NETWORK
TITLE = ---- ---- Recoger el Atributo de las UTs - PILA (La Carga es una Pila)
/////////////////////////////////////////////////////////////////////////
/////////////////////////////////////////////////////////////////////////
/////////////////////////////////////////////////////////////////////////
AtributoDeUTs_PILA:NOP   0;
      +AR2  P#5.0;

      OPN   DB [#DBEventosRec];
      L     DBB [AR2, P#0.0];  // Sacar el Valor del Campo
      T     #Leido;
      +AR2  P#1.0;

      L     #Leido;  // Comparar si es cero
      L     '0';  // La Carga No es Pila
      ==I;
      JC    InicioBucleAtributos_EventosDeLasUTs;

      SET;
      S     #AtributosDeUTs.AtributosTipoDeCarga.Pila;


// Continuo con el Evento
      JU    InicioBucleAtributos_EventosDeLasUTs;



NETWORK
TITLE = ---- ---- Recoger el Atributo de las UTs - VACI ( La carga esta vacia de contenido)
/////////////////////////////////////////////////////////////////////////
/////////////////////////////////////////////////////////////////////////
/////////////////////////////////////////////////////////////////////////
AtributoDeUTs_VACI:NOP   0;
      +AR2  P#5.0;

      OPN   DB [#DBEventosRec];
      L     DBB [AR2, P#0.0];  // Sacar el Valor del Campo
      T     #Leido;
      +AR2  P#1.0;

      L     #Leido;  // Comparar si es cero
      L     '0';  // La carga No esta Vacia
      ==I;
      JC    InicioBucleAtributos_EventosDeLasUTs;

      SET;
      S     #AtributosDeUTs.AtributosTipoDeCarga.Vacia;


// Continuo con el Evento
      JU    InicioBucleAtributos_EventosDeLasUTs;



NETWORK
TITLE = ---- ---- Recoger el Atributo de las UTs - COTA ( Cota de Altura)
/////////////////////////////////////////////////////////////////////////
/////////////////////////////////////////////////////////////////////////
/////////////////////////////////////////////////////////////////////////
AtributoDeUTs_COTA:NOP   0;
      +AR2  P#5.0;
      TAR2;
      T     #P_Eventos;
      SRD   3;
      T     #OffsetInicial;

// Obtener el Valor del Atributo
      CALL  "FC892_Obtener_ValorDelAtributo"
      ( DB_String := #DBEventosRec,
        OffsetIni := #OffsetInicial,
        Valor     := #ValorDeAtributo
      );

      L     #ValorDeAtributo;  // Lo guardo
      T     #AtributosDeUTs.CotaAltura;

// Continuo con el Evento
      L     #P_Eventos;
      LAR2;
      JU    InicioBucleAtributos_EventosDeLasUTs;



NETWORK
TITLE = ---- ---- Recoger el Atributo de las UTs - COTW (Cota de Anchura)
/////////////////////////////////////////////////////////////////////////
/////////////////////////////////////////////////////////////////////////
/////////////////////////////////////////////////////////////////////////
AtributoDeUTs_COTW:NOP   0;
      +AR2  P#5.0;
      TAR2;
      T     #P_Eventos;
      SRD   3;
      T     #OffsetInicial;

// Obtener el Valor del Atributo
      CALL  "FC892_Obtener_ValorDelAtributo"
      ( DB_String := #DBEventosRec,
        OffsetIni := #OffsetInicial,
        Valor     := #ValorDeAtributo
      );

      L     #ValorDeAtributo;  // Lo guardo
      T     #AtributosDeUTs.CotaAnchura;

// Continuo con el Evento
      L     #P_Eventos;
      LAR2;
      JU    InicioBucleAtributos_EventosDeLasUTs;



NETWORK
TITLE = ---- ---- Recoger el Atributo de las UTs - COTL (Cota de Profundidad)
/////////////////////////////////////////////////////////////////////////
/////////////////////////////////////////////////////////////////////////
/////////////////////////////////////////////////////////////////////////
AtributoDeUTs_COTL:NOP   0;
      +AR2  P#5.0;
      TAR2;
      T     #P_Eventos;
      SRD   3;
      T     #OffsetInicial;

// Obtener el Valor del Atributo
      CALL  "FC892_Obtener_ValorDelAtributo"
      ( DB_String := #DBEventosRec,
        OffsetIni := #OffsetInicial,
        Valor     := #ValorDeAtributo
      );

      L     #ValorDeAtributo;  // Lo guardo
      T     #AtributosDeUTs.CotaProfundidad;

// Continuo con el Evento
      L     #P_Eventos;
      LAR2;
      JU    InicioBucleAtributos_EventosDeLasUTs;



NETWORK
TITLE = ---- ---- Recoger el Atributo de las UTs - PESO
/////////////////////////////////////////////////////////////////////////
/////////////////////////////////////////////////////////////////////////
/////////////////////////////////////////////////////////////////////////
AtributoDeUTs_PESO:NOP   0;
      +AR2  P#5.0;
      TAR2;
      T     #P_Eventos;
      SRD   3;
      T     #OffsetInicial;

// Obtener el Valor del Atributo
      CALL  "FC892_Obtener_ValorDelAtributo"
      ( DB_String := #DBEventosRec,
        OffsetIni := #OffsetInicial,
        Valor     := #ValorDeAtributo
      );

      L     #ValorDeAtributo;  // Lo guardo
      T     #AtributosDeUTs.Peso;

// Continuo con el Evento
      L     #P_Eventos;
      LAR2;
      JU    InicioBucleAtributos_EventosDeLasUTs;



NETWORK
TITLE = ---- ---- Recoger el Atributo de las UTs - ALTO (Codigo de Altura)
/////////////////////////////////////////////////////////////////////////
/////////////////////////////////////////////////////////////////////////
/////////////////////////////////////////////////////////////////////////
AtributoDeUTs_ALTO:NOP   0;
      +AR2  P#5.0;
      TAR2;
      T     #P_Eventos;
      SRD   3;
      T     #OffsetInicial;

// Obtener el Valor del Atributo
      CALL  "FC892_Obtener_ValorDelAtributo"
      ( DB_String := #DBEventosRec,
        OffsetIni := #OffsetInicial,
        Valor     := #ValorDeAtributo
      );

      L     #ValorDeAtributo;  // Lo guardo
      T     #AtributosDeUTs.GaliboAltura;

// Continuo con el Evento
      L     #P_Eventos;
      LAR2;
      JU    InicioBucleAtributos_EventosDeLasUTs;



NETWORK
TITLE = ---- ---- Recoger el Atributo de las UTs - ANCH (Codigo de Anchura)
/////////////////////////////////////////////////////////////////////////
/////////////////////////////////////////////////////////////////////////
/////////////////////////////////////////////////////////////////////////
AtributoDeUTs_ANCH:NOP   0;
      +AR2  P#5.0;
      TAR2;
      T     #P_Eventos;
      SRD   3;
      T     #OffsetInicial;

// Obtener el Valor del Atributo
      CALL  "FC892_Obtener_ValorDelAtributo"
      ( DB_String := #DBEventosRec,
        OffsetIni := #OffsetInicial,
        Valor     := #ValorDeAtributo
      );

      L     #ValorDeAtributo;  // Lo guardo
      T     #AtributosDeUTs.GaliboAnchura;

// Continuo con el Evento
      L     #P_Eventos;
      LAR2;
      JU    InicioBucleAtributos_EventosDeLasUTs;



NETWORK
TITLE = ---- ---- Recoger el Atributo de las UTs - PROF (Codigo de Profundidad)
/////////////////////////////////////////////////////////////////////////
/////////////////////////////////////////////////////////////////////////
/////////////////////////////////////////////////////////////////////////
AtributoDeUTs_PROF:NOP   0;
      +AR2  P#5.0;
      TAR2;
      T     #P_Eventos;
      SRD   3;
      T     #OffsetInicial;

// Obtener el Valor del Atributo
      CALL  "FC892_Obtener_ValorDelAtributo"
      ( DB_String := #DBEventosRec,
        OffsetIni := #OffsetInicial,
        Valor     := #ValorDeAtributo
      );

      L     #ValorDeAtributo;  // Lo guardo
      T     #AtributosDeUTs.GaliboProfundidad;

// Continuo con el Evento
      L     #P_Eventos;
      LAR2;
      JU    InicioBucleAtributos_EventosDeLasUTs;



NETWORK
TITLE = ---- ---- Recoger el Atributo de las UTs - TACO (Codigo de Taco)
/////////////////////////////////////////////////////////////////////////
/////////////////////////////////////////////////////////////////////////
/////////////////////////////////////////////////////////////////////////
AtributoDeUTs_TACO:NOP   0;
      +AR2  P#5.0;
      TAR2;
      T     #P_Eventos;
      SRD   3;
      T     #OffsetInicial;

// Obtener el Valor del Atributo
      CALL  "FC892_Obtener_ValorDelAtributo"
      ( DB_String := #DBEventosRec,
        OffsetIni := #OffsetInicial,
        Valor     := #ValorDeAtributo
      );

      L     #ValorDeAtributo;  // Lo guardo
      T     #AtributosDeUTs.GaliboTaco;

// Continuo con el Evento
      L     #P_Eventos;
      LAR2;
      JU    InicioBucleAtributos_EventosDeLasUTs;



NETWORK
TITLE = ---- ---- Recoger el Atributo de las UTs - HUEC (Codigo de Hueco)
/////////////////////////////////////////////////////////////////////////
/////////////////////////////////////////////////////////////////////////
/////////////////////////////////////////////////////////////////////////
AtributoDeUTs_HUEC:NOP   0;
      +AR2  P#5.0;
      TAR2;
      T     #P_Eventos;
      SRD   3;
      T     #OffsetInicial;

// Obtener el Valor del Atributo
      CALL  "FC892_Obtener_ValorDelAtributo"
      ( DB_String := #DBEventosRec,
        OffsetIni := #OffsetInicial,
        Valor     := #ValorDeAtributo
      );

      L     #ValorDeAtributo;  // Lo guardo
      T     #AtributosDeUTs.GaliboHueco;

// Continuo con el Evento
      L     #P_Eventos;
      LAR2;
      JU    InicioBucleAtributos_EventosDeLasUTs;



NETWORK
TITLE = ---- ---- Recoger el Atributo de las UTs - HUER (Codigo de Hueco de Remontada)
/////////////////////////////////////////////////////////////////////////
/////////////////////////////////////////////////////////////////////////
/////////////////////////////////////////////////////////////////////////
AtributoDeUTs_HUER:NOP   0;
      +AR2  P#5.0;
      TAR2;
      T     #P_Eventos;
      SRD   3;
      T     #OffsetInicial;

// Obtener el Valor del Atributo
      CALL  "FC892_Obtener_ValorDelAtributo"
      ( DB_String := #DBEventosRec,
        OffsetIni := #OffsetInicial,
        Valor     := #ValorDeAtributo
      );

      L     #ValorDeAtributo;  // Lo guardo
      T     #AtributosDeUTs.GaliboHuecoRemontada;

// Continuo con el Evento
      L     #P_Eventos;
      LAR2;
      JU    InicioBucleAtributos_EventosDeLasUTs;



NETWORK
TITLE = ---- ---- Recoger el Atributo de las UTs - COLO (Codigo de Color)
/////////////////////////////////////////////////////////////////////////
/////////////////////////////////////////////////////////////////////////
/////////////////////////////////////////////////////////////////////////
AtributoDeUTs_COLO:NOP   0;
      +AR2  P#5.0;

      OPN   DB [#DBEventosRec];
      L     DBD [AR2, P#0.0];
      T     #EtiquetaAtributo;

// Obtener el Valor del Atributo
      CALL  "FC894_Obtener_ValorDeEtiqueta"
      ( EtiquetaEvento := #EtiquetaAtributo,
        ValorEvento    := #ValorDeEtiqueta
      );

      L     #ValorDeEtiqueta;  // Lo guardo
      T     #AtributosDeUTs.GaliboColor;

// Continuo con el Evento
      +AR2  P#4.0;
      JU    InicioBucleAtributos_EventosDeLasUTs;



NETWORK
TITLE = ---- ---- Recoger el Atributo de las UTs - PATI (Codigo de Patin)
/////////////////////////////////////////////////////////////////////////
/////////////////////////////////////////////////////////////////////////
/////////////////////////////////////////////////////////////////////////
AtributoDeUTs_PATI:NOP   0;
      +AR2  P#5.0;
      TAR2;
      T     #P_Eventos;
      SRD   3;
      T     #OffsetInicial;

// Obtener el Valor del Atributo
      CALL  "FC892_Obtener_ValorDelAtributo"
      ( DB_String := #DBEventosRec,
        OffsetIni := #OffsetInicial,
        Valor     := #ValorDeAtributo
      );

      L     #ValorDeAtributo;  // Lo guardo
      T     #AtributosDeUTs.GaliboPatin;

// Continuo con el Evento
      L     #P_Eventos;
      LAR2;
      JU    InicioBucleAtributos_EventosDeLasUTs;



NETWORK
TITLE = ---- ---- Recoger el Atributo de las UTs - LETI (Lado de la Etiqueta)
/////////////////////////////////////////////////////////////////////////
/////////////////////////////////////////////////////////////////////////
/////////////////////////////////////////////////////////////////////////
AtributoDeUTs_LETI:NOP   0;
      +AR2  P#5.0;
      TAR2;
      T     #P_Eventos;
      SRD   3;
      T     #OffsetInicial;

// Obtener el Valor del Atributo
      CALL  "FC892_Obtener_ValorDelAtributo"
      ( DB_String := #DBEventosRec,
        OffsetIni := #OffsetInicial,
        Valor     := #ValorDeAtributo
      );

      L     #ValorDeAtributo;  // Lo guardo
      L     1;
      +I;
      T     #AtributosDeUTs.PosicionDeLaEtiqueta;

// Continuo con el Evento
      L     #P_Eventos;
      LAR2;
      JU    InicioBucleAtributos_EventosDeLasUTs;



NETWORK
TITLE = ---- ---- Recoger el Atributo de las UTs - SGAP ( SGA - Error de Peso)
/////////////////////////////////////////////////////////////////////////
/////////////////////////////////////////////////////////////////////////
/////////////////////////////////////////////////////////////////////////
AtributoDeUTs_SGAP:NOP   0;
      +AR2  P#5.0;

      OPN   DB [#DBEventosRec];
      L     DBW [AR2, P#0.0];
      T     #Leido;

      L     0;  // Por defecto No Error
      T     #ValorDeAtributo;

      L     'NO';  // Tiene Error ?
      L     #Leido;
      ==I;
      JC    AtributoDeUTs_SGAP_NoError;

      L     W#16#08;
      T     #ValorDeAtributo;

AtributoDeUTs_SGAP_NoError:NOP   0;
      L     #ValorDeAtributo;
      L     #AtributosDeUTs.GaliboSGA;
      +I;
      T     #AtributosDeUTs.GaliboSGA;

// Continuo con el Evento
      +AR2  P#2.0;
      JU    InicioBucleAtributos_EventosDeLasUTs;



NETWORK
TITLE = ---- ---- Recoger el Atributo de las UTs - SGAE ( SGA - Error de Etiqueta)
/////////////////////////////////////////////////////////////////////////
/////////////////////////////////////////////////////////////////////////
/////////////////////////////////////////////////////////////////////////
AtributoDeUTs_SGAE:NOP   0;
      +AR2  P#5.0;

      OPN   DB [#DBEventosRec];
      L     DBW [AR2, P#0.0];
      T     #Leido;

      L     0;  // Por defecto No Error
      T     #ValorDeAtributo;

      L     'NO';  // Tiene Error ?
      L     #Leido;
      ==I;
      JC    AtributoDeUTs_SGAE_NoError;

      L     W#16#04;
      T     #ValorDeAtributo;

AtributoDeUTs_SGAE_NoError:NOP   0;
      L     #ValorDeAtributo;
      L     #AtributosDeUTs.GaliboSGA;
      +I;
      T     #AtributosDeUTs.GaliboSGA;

// Continuo con el Evento
      +AR2  P#2.0;
      JU    InicioBucleAtributos_EventosDeLasUTs;



NETWORK
TITLE = ---- ---- Recoger el Atributo de las UTs - SGAD ( SGA - Error de Dimensiones)
/////////////////////////////////////////////////////////////////////////
/////////////////////////////////////////////////////////////////////////
/////////////////////////////////////////////////////////////////////////
AtributoDeUTs_SGAD:NOP   0;
      +AR2  P#5.0;

      OPN   DB [#DBEventosRec];
      L     DBW [AR2, P#0.0];
      T     #Leido;

      L     0;  // Por defecto No Error
      T     #ValorDeAtributo;

      L     'NO';  // Tiene Error ?
      L     #Leido;
      ==I;
      JC    AtributoDeUTs_SGAD_NoError;

      L     W#16#02;
      T     #ValorDeAtributo;

AtributoDeUTs_SGAD_NoError:NOP   0;
      L     #ValorDeAtributo;
      L     #AtributosDeUTs.GaliboSGA;
      +I;
      T     #AtributosDeUTs.GaliboSGA;

// Continuo con el Evento
      +AR2  P#2.0;
      JU    InicioBucleAtributos_EventosDeLasUTs;



NETWORK
TITLE = ---- ---- Recoger el Atributo de las UTs - SGA_ ( SGA - Error General)
/////////////////////////////////////////////////////////////////////////
/////////////////////////////////////////////////////////////////////////
/////////////////////////////////////////////////////////////////////////
AtributoDeUTs_SGA_Error:NOP   0;
      +AR2  P#5.0;

      OPN   DB [#DBEventosRec];
      L     DBW [AR2, P#0.0];
      T     #Leido;

      L     0;  // Por defecto No Error
      T     #ValorDeAtributo;

      L     'NO';  // Tiene Error ?
      L     #Leido;
      ==I;
      JC    AtributoDeUTs_SGA_Error_NoError;

      L     W#16#01;
      T     #ValorDeAtributo;

AtributoDeUTs_SGA_Error_NoError:NOP   0;
      L     #ValorDeAtributo;
      L     #AtributosDeUTs.GaliboSGA;
      +I;
      T     #AtributosDeUTs.GaliboSGA;

// Continuo con el Evento
      +AR2  P#2.0;
      JU    InicioBucleAtributos_EventosDeLasUTs;



NETWORK
TITLE = ---- ---- Recoger el Atributo de las UTs - RSLT (Mover UT - Resultado)
/////////////////////////////////////////////////////////////////////////
/////////////////////////////////////////////////////////////////////////
/////////////////////////////////////////////////////////////////////////
AtributoDeUTs_RSLT:NOP   0;
      +AR2  P#5.0;

      OPN   DB [#DBEventosRec];
      L     DBW [AR2, P#0.0];  // Sacar el Valor del Campo
      T     #Leido;

      SET;  // Inicializar a NOK
      S     #AtributosDeUTs.CambiarUTDeMesa.NOK;
      R     #AtributosDeUTs.CambiarUTDeMesa.OK;

      L     #Leido;  // Comparar si es NO ?
      L     'SI';
      <>I;
      JC    InicioBucleAtributos_EventosDeLasUTs;

      SET;  // Inicializar a OK
      R     #AtributosDeUTs.CambiarUTDeMesa.NOK;
      S     #AtributosDeUTs.CambiarUTDeMesa.OK;

// Continuo con el Evento
      +AR2  P#2.0;
      JU    InicioBucleAtributos_EventosDeLasUTs;



NETWORK
TITLE = ---- ---- Recoger el Atributo de las UTs - PDST (Mover UT - Posicion en la Cola de Mesa)
/////////////////////////////////////////////////////////////////////////
/////////////////////////////////////////////////////////////////////////
/////////////////////////////////////////////////////////////////////////
AtributoDeUTs_PDST:NOP   0;
      +AR2  P#5.0;

      OPN   DB [#DBEventosRec];
      L     DBD [AR2, P#0.0];  // Sacar el Valor del Campo
      T     #EtiquetaAtributo;

      SET;  // Inicializar a Final
      S     #AtributosDeUTs.CambiarUTDeMesa.Final;
      R     #AtributosDeUTs.CambiarUTDeMesa.Inicio;

      L     #EtiquetaAtributo;  // Comparar si es _FIN ?
      L     '_INI';
      <>D;
      JC    InicioBucleAtributos_EventosDeLasUTs;

      SET;  // Inicializar a Inicio
      R     #AtributosDeUTs.CambiarUTDeMesa.Final;
      S     #AtributosDeUTs.CambiarUTDeMesa.Inicio;

// Continuo con el Evento
      +AR2  P#4.0;
      JU    InicioBucleAtributos_EventosDeLasUTs;



NETWORK
TITLE = ---- ---- Recoger el Atributo de las UTs - DEST (Mover UT - Destino)
/////////////////////////////////////////////////////////////////////////
/////////////////////////////////////////////////////////////////////////
/////////////////////////////////////////////////////////////////////////
AtributoDeUTs_DEST:NOP   0;
      +AR2  P#5.0;
      TAR2;
      T     #P_Eventos;
      SRD   3;
      T     #OffsetInicial;

// Obtener el Valor del Atributo
      CALL  "FC892_Obtener_ValorDelAtributo"
      ( DB_String := #DBEventosRec,
        OffsetIni := #OffsetInicial,
        Valor     := #ValorDeAtributo
      );

      L     #ValorDeAtributo;  // Lo guardo
      L     #AtributosDeUTs.CambiarUTDeMesa.Destino;

// Continuo con el Evento
      L     #P_Eventos;
      LAR2;
      JU    InicioBucleAtributos_EventosDeLasUTs;



NETWORK
TITLE = ////////////////////////////////////////////////////////////////////////////////////////////////////////////

NETWORK
TITLE = Analizar la lista de los Atributos de los Dispositivos
Atributos_EventosDeLosDispositivos:NOP   0;

/////////////////////////////////////////////////////////////////////////
/////////////////////////////////////////////////////////////////////////
/////////////////////////////////////////////////////////////////////////
// Inicializa variables de los Atributos de las UTs
      L     0;
      T     #Cero;

      CALL  FILL
      ( BVAL    := #Cero,
        RET_VAL := #ReturnValor,
        BLK     := #AtributosDeDispositivos
      );  // Inicializa Atributos de las UTS



NETWORK
TITLE = ----
/////////////////////////////////////////////////////////////////////////
/////////////////////////////////////////////////////////////////////////
// Buscando Atributos o Final del Evento
      +AR2  P#4.0;  // Prepara Puntero para ver los atributos

InicioBucleAtributos_EventosDeLosDispositivos:NOP   0;
      OPN   DB [#DBEventosRec];
      L     DBB [AR2, P#0.0];
      T     #Leido;

// Inicio de atributo - Ir a tratar los atributos
      L     #Leido;
      L     '[';  // '[' - Inicio de Atributo
      ==I;  // Atributo del Evento
      JC    EncontradoAtributos_EventosDeLosDispositivos;

// Fin del Evento
      L     #Leido;
      L     '}';  // '}' - Fin del Evento
      ==I;  // Se acabo el evento
      JC    FinalAtributos_EventosDeLosDispositivos;

      +AR2  P#1.0;  // Seguir buscado atributo
      JU    InicioBucleAtributos_EventosDeLosDispositivos;


/////////////////////////////////////////////////////////////////////////
/////////////////////////////////////////////////////////////////////////
// Se acaba el Evento - Ir a guardar datos del Evento
FinalAtributos_EventosDeLosDispositivos:NOP   0;
      TAR2;
      T     #P_Eventos;  // Guardo Por donde voy en la lista de eventos
      JU    GuardarDatos_EventosRecibidos;



NETWORK
TITLE = Distribucion de los Atributos de los DIspositivos (LIsta del DB de Conversion)
EncontradoAtributos_EventosDeLosDispositivos:NOP   0;

/////////////////////////////////////////////////////////////////////////
/////////////////////////////////////////////////////////////////////////
/////////////////////////////////////////////////////////////////////////
/////////////////////////////////////////////////////////////////////////
// Mirar que Atributo del Evento  es ?
      +AR2  P#1.0;
      OPN   DB [#DBEventosRec];
      L     DBD [AR2, P#0.0];  // Atributo - 4 Caracteres
      T     #Atributo;

/////////////////////////////////////////////////////////////////////////
/////////////////////////////////////////////////////////////////////////
/////////////////////////////////////////////////////////////////////////
// Buscar numero de Atributo
      L     1;
      T     #NumeroAtributo;
BucleDeBusqueda_NumeroDeAtributoDeDispositivos:NOP   0;

// -- Se ha encontrado el Atributo Recibido
      L     "DB870_ConversorEventos".AtributosRecibidosDeDispositivos[#NumeroAtributo];
      L     #Atributo;
      ==D;
      JC    Encontrado_NumeroDeAtributoDeDispositivos;

// -- Final de la lista de Atributo Recibidos - No Encontrado
      L     "DB870_ConversorEventos".AtributosRecibidosDeDispositivos[#NumeroAtributo];
      L     0;
      ==D;
      JC    InicioBucleAtributos_EventosDeLosDispositivos;

// --- Maximo del Array de la Lista de Atributo Recibidos - No Encontrado
      L     #NumeroAtributo;
      L     "CTE_MaxArrayConversion";
      >=I;
      JC    InicioBucleAtributos_EventosDeLosDispositivos;


// --- Continuar la Busqueda
      L     #NumeroAtributo;
      L     1;
      +I;
      T     #NumeroAtributo;
      JU    BucleDeBusqueda_NumeroDeAtributoDeDispositivos;



NETWORK
TITLE = ----
/////////////////////////////////////////////////////////////////////////
/////////////////////////////////////////////////////////////////////////
/////////////////////////////////////////////////////////////////////////
// Distribuir dependiendo del Resultado de la Busqueda de Atributo Recibido
Encontrado_NumeroDeAtributoDeDispositivos:NOP   0;
      L     #NumeroAtributo;
      JL    NoExiste_NumeroDeAtibutoDeDispositivos;

      JU    NoExiste_NumeroDeAtibutoDeDispositivos;
      JU    AtributoDeDispositivos_TIPO;  // Atributo (01) - TIPO
      JU    AtributoDeDispositivos_NUME;  // Atributo (02) - NUME
      JU    AtributoDeDispositivos_NUES;  // Atributo (03) - NUES
      JU    AtributoDeDispositivos_HABI;  // Atributo (04) - HABI
      JU    AtributoDeDispositivos_PRIO;  // Atributo (05) - PRIO

      JU    AtributoDeDispositivos_SONO;  // Atributo (06) - SONO
      JU    AtributoDeDispositivos_VERD;  // Atributo (07) - VERD
      JU    AtributoDeDispositivos_ROJO;  // Atributo (08) - ROJO
      JU    AtributoDeDispositivos_AMAR;  // Atributo (09) - AMAR
      JU    AtributoDeDispositivos_AZUL;  // Atributo (10) - AZUL

      JU    AtributoDeDispositivos_MOTI;  // Atributo (11) - MOTI
      JU    AtributoDeDispositivos_OPER;  // Atributo (12) - OPER
      JU    AtributoDeDispositivos_TEXT;  // Atributo (13) - TEXT

      JU    AtributoDeDispositivos_HORQ;  // Atributo (14) - HORQ
      JU    AtributoDeDispositivos_POSI;  // Atributo (15) - POSI

/////////////////////////////////////////////////////////////////////////
NoExiste_NumeroDeAtibutoDeDispositivos:NOP   0;
      JU    InicioBucleAtributos_EventosDeLosDispositivos;



NETWORK
TITLE = ---- ---- Recoger el Atributo de los Dispositivos - TIPO
/////////////////////////////////////////////////////////////////////////
/////////////////////////////////////////////////////////////////////////
/////////////////////////////////////////////////////////////////////////
AtributoDeDispositivos_TIPO:NOP   0;
      +AR2  P#5.0;

      OPN   DB [#DBEventosRec];
      L     DBD [AR2, P#0.0];
      T     #EtiquetaAtributo;

// Obtener el Valor del Tipo de Dispositivo

      CALL  "FC894_Obtener_ValorDeEtiqueta"
      ( EtiquetaEvento := #EtiquetaAtributo,
        ValorEvento    := #ValorDeEtiqueta
      );

      L     #ValorDeEtiqueta;  // Lo guardo
      T     #AtributosDeDispositivos.Tipo;

// Continuo con el Evento
      +AR2  P#4.0;
      JU    InicioBucleAtributos_EventosDeLosDispositivos;



NETWORK
TITLE = ---- ---- Recoger el Atributo de los Dispositivos - NUME
/////////////////////////////////////////////////////////////////////////
/////////////////////////////////////////////////////////////////////////
/////////////////////////////////////////////////////////////////////////
AtributoDeDispositivos_NUME:NOP   0;
      +AR2  P#5.0;
      TAR2;
      T     #P_Eventos;
      SRD   3;
      T     #OffsetInicial;

// Obtener el Valor del Numero del Dispositivo

      CALL  "FC892_Obtener_ValorDelAtributo"
      ( DB_String := #DBEventosRec,
        OffsetIni := #OffsetInicial,
        Valor     := #ValorDeAtributo
      );
      L     #ValorDeAtributo;  // Lo guardo
      T     #AtributosDeDispositivos.Numero;

// Continuo con el Evento
      L     #P_Eventos;
      LAR2;
      JU    InicioBucleAtributos_EventosDeLosDispositivos;



NETWORK
TITLE = ---- ---- Recoger el Atributo de los Dispositivos - NUES (Nuevo Estado)
/////////////////////////////////////////////////////////////////////////
/////////////////////////////////////////////////////////////////////////
/////////////////////////////////////////////////////////////////////////
AtributoDeDispositivos_NUES:NOP   0;
      +AR2  P#5.0;

      OPN   DB [#DBEventosRec];
      L     DBD [AR2, P#0.0];
      T     #EtiquetaAtributo;

// Obtener el Valor del Tipo de Dispositivo
      CALL  "FC894_Obtener_ValorDeEtiqueta"
      ( EtiquetaEvento := #EtiquetaAtributo,
        ValorEvento    := #ValorDeEtiqueta
      );

      L     #ValorDeEtiqueta;  // Lo guardo
      T     #AtributosDeDispositivos.NuevoEstado;

// Continuo con el Evento
      +AR2  P#4.0;
      JU    InicioBucleAtributos_EventosDeLosDispositivos;



NETWORK
TITLE = ---- ---- Recoger el Atributo de los Dispositivos - HABI
/////////////////////////////////////////////////////////////////////////
/////////////////////////////////////////////////////////////////////////
/////////////////////////////////////////////////////////////////////////
AtributoDeDispositivos_HABI:NOP   0;
      +AR2  P#5.0;

      OPN   DB [#DBEventosRec];
      L     DBW [AR2, P#0.0];
      T     #Leido;

      L     2001;
      T     #ValorDeAtributo;

      L     #Leido;
      L     'NO';
      ==I;
      JCN   AtributoDeDispositivos_HABI_NoHabilitar;

      L     2002;
      T     #ValorDeAtributo;

AtributoDeDispositivos_HABI_NoHabilitar:NOP   0;
      L     #ValorDeAtributo;  // Lo guardo
      T     #AtributosDeDispositivos.Habilitado;

// Continuo con el Evento
      +AR2  P#2.0;
      JU    InicioBucleAtributos_EventosDeLosDispositivos;



NETWORK
TITLE = ---- ---- Recoger el Atributo de los Dispositivos - PRIO
/////////////////////////////////////////////////////////////////////////
/////////////////////////////////////////////////////////////////////////
/////////////////////////////////////////////////////////////////////////
AtributoDeDispositivos_PRIO:NOP   0;
      +AR2  P#5.0;
      TAR2;
      T     #P_Eventos;
      SRD   3;
      T     #OffsetInicial;

// Obtener el Valor del Numero del Dispositivo
      CALL  "FC892_Obtener_ValorDelAtributo"
      ( DB_String := #DBEventosRec,
        OffsetIni := #OffsetInicial,
        Valor     := #ValorDeAtributo
      );

      L     #ValorDeAtributo;  // Lo guardo
      L     1;
      +I;
      T     #AtributosDeDispositivos.Prioridad;

// Continuo con el Evento
      L     #P_Eventos;
      LAR2;
      JU    InicioBucleAtributos_EventosDeLosDispositivos;



NETWORK
TITLE = ---- ---- Recoger el Atributo de los Dispositivos - SONO (Baliza - Sirena)
/////////////////////////////////////////////////////////////////////////
/////////////////////////////////////////////////////////////////////////
/////////////////////////////////////////////////////////////////////////
AtributoDeDispositivos_SONO:NOP   0;
      +AR2  P#5.0;

      SET;
      S     #AtributosDeDispositivos.BalizaColor.Sonoro;


// Continuo con el Evento
      JU    InicioBucleAtributos_EventosDeLosDispositivos;



NETWORK
TITLE = ---- ---- Recoger el Atributo de los Dispositivos - VERD (Baliza - Verde)
/////////////////////////////////////////////////////////////////////////
/////////////////////////////////////////////////////////////////////////
/////////////////////////////////////////////////////////////////////////
AtributoDeDispositivos_VERD:NOP   0;
      +AR2  P#5.0;

      SET;
      S     #AtributosDeDispositivos.BalizaColor.Verde;


// Continuo con el Evento
      JU    InicioBucleAtributos_EventosDeLosDispositivos;



NETWORK
TITLE = ---- ---- Recoger el Atributo de los Dispositivos - ROJO (Baliza - Roja)
/////////////////////////////////////////////////////////////////////////
/////////////////////////////////////////////////////////////////////////
/////////////////////////////////////////////////////////////////////////
AtributoDeDispositivos_ROJO:NOP   0;
      +AR2  P#5.0;

      SET;
      S     #AtributosDeDispositivos.BalizaColor.Rojo;


// Continuo con el Evento
      JU    InicioBucleAtributos_EventosDeLosDispositivos;



NETWORK
TITLE = ---- ---- Recoger el Atributo de los Dispositivos - AMAR (Baliza - Amarilla)
/////////////////////////////////////////////////////////////////////////
/////////////////////////////////////////////////////////////////////////
/////////////////////////////////////////////////////////////////////////
AtributoDeDispositivos_AMAR:NOP   0;
      +AR2  P#5.0;

      SET;
      S     #AtributosDeDispositivos.BalizaColor.Amarillo;


// Continuo con el Evento
      JU    InicioBucleAtributos_EventosDeLosDispositivos;



NETWORK
TITLE = ---- ---- Recoger el Atributo de los Dispositivos - AZUL (Baliza - Azul)
/////////////////////////////////////////////////////////////////////////
/////////////////////////////////////////////////////////////////////////
/////////////////////////////////////////////////////////////////////////
AtributoDeDispositivos_AZUL:NOP   0;
      +AR2  P#5.0;

      SET;
      S     #AtributosDeDispositivos.BalizaColor.Azul;


// Continuo con el Evento
      JU    InicioBucleAtributos_EventosDeLosDispositivos;



NETWORK
TITLE = ---- ---- Recoger el Atributo de los Dispositivos - MOTI (Moitvo del Envio a Error del JdT )
/////////////////////////////////////////////////////////////////////////
/////////////////////////////////////////////////////////////////////////
/////////////////////////////////////////////////////////////////////////
AtributoDeDispositivos_MOTI:NOP   0;
      +AR2  P#5.0;

// - Recorrer el Motivo del Error es una STRING
      L     2;  // Inicializaciones
      T     #LonguitudTextoRecibido;

// Inicio a Recoger el Motivo del Error
AtributoDeDispositivos_MOTI_InicioBucle:NOP   0;
      OPN   DB [#DBEventosRec];
      L     DBB [AR2, P#0.0];  // Leer ek texto
      T     #Leido;

      L     #Leido;  // Es final del Texto
      L     '[';
      ==I;
      JC    AtributoDeDispositivos_MOTI_FinalBucle;

      L     #Leido;  // Es final del Texto
      L     '}';
      ==I;
      JC    AtributoDeDispositivos_MOTI_FinalBucle;

      L     #Leido;  // Guardo el texto
      T     #AtributosDeDispositivos.MotivoDelError[#LonguitudTextoRecibido];

// Incremetar punteros
      +AR2  P#1.0;
      L     #LonguitudTextoRecibido;
      L     1;
      +I;
      T     #LonguitudTextoRecibido;

      L     0;  // Pongo el siguiente a cero
      T     #AtributosDeDispositivos.MotivoDelError[#LonguitudTextoRecibido];

      JU    AtributoDeDispositivos_MOTI_InicioBucle;


// - Continuo con el Evento
AtributoDeDispositivos_MOTI_FinalBucle:NOP   0;
      L     48;  // Inicio la carcacteristica de la STRING
      T     #AtributosDeDispositivos.MotivoDelError[0];
      L     #LonguitudTextoRecibido;
      L     2;
      -I;
      T     #AtributosDeDispositivos.MotivoDelError[1];

      JU    InicioBucleAtributos_EventosDeLosDispositivos;



NETWORK
TITLE = ---- ---- Recoger el Atributo de los Dispositivos - OPER (Operacion a realizar de las Maquinas)
/////////////////////////////////////////////////////////////////////////
/////////////////////////////////////////////////////////////////////////
/////////////////////////////////////////////////////////////////////////
AtributoDeDispositivos_OPER:NOP   0;
      +AR2  P#5.0;

      OPN   DB [#DBEventosRec];
      L     DBD [AR2, P#0.0];
      T     #EtiquetaAtributo;

// Obtener el Valor del Tipo de Dispositivo
      CALL  "FC894_Obtener_ValorDeEtiqueta"
      ( EtiquetaEvento := #EtiquetaAtributo,
        ValorEvento    := #ValorDeEtiqueta
      );

      L     #ValorDeEtiqueta;  // Lo guardo
      T     #AtributosDeDispositivos.Operacion;

// Continuo con el Evento
      +AR2  P#4.0;
      JU    InicioBucleAtributos_EventosDeLosDispositivos;



NETWORK
TITLE = ---- ---- Recoger el Atributo de los Dispositivos - TEXT
/////////////////////////////////////////////////////////////////////////
/////////////////////////////////////////////////////////////////////////
/////////////////////////////////////////////////////////////////////////
AtributoDeDispositivos_TEXT:NOP   0;
      +AR2  P#5.0;

// - Recorrer el Motivo del Error es una STRING
      L     2;  // Inicializaciones
      T     #LonguitudTextoRecibido;

// Inicio a Recoger el Texto
AtributoDeDispositivos_TEXT_InicioBucle:NOP   0;
      OPN   DB [#DBEventosRec];
      L     DBB [AR2, P#0.0];  // Leer ek texto
      T     #Leido;

      L     #Leido;  // Es final del Texto
      L     '[';
      ==I;
      JC    AtributoDeDispositivos_TEXT_FinalBucle;

      L     #Leido;  // Es final del Texto
      L     '}';
      ==I;
      JC    AtributoDeDispositivos_TEXT_FinalBucle;

      L     #Leido;  // Guardo el texto
      T     #AtributosDeDispositivos.TextoRecibido[#LonguitudTextoRecibido];

// Incremetar punteros
      +AR2  P#1.0;
      L     #LonguitudTextoRecibido;
      L     1;
      +I;
      T     #LonguitudTextoRecibido;

      L     0;  // Pongo el siguiente a cero
      T     #AtributosDeDispositivos.TextoRecibido[#LonguitudTextoRecibido];

      JU    AtributoDeDispositivos_TEXT_InicioBucle;


// - Continuo con el Evento
AtributoDeDispositivos_TEXT_FinalBucle:NOP   0;
      L     48;  // Inicio la carcacteristica de la STRING
      T     #AtributosDeDispositivos.TextoRecibido[0];
      L     #LonguitudTextoRecibido;
      L     2;
      -I;
      T     #AtributosDeDispositivos.TextoRecibido[1];

      JU    InicioBucleAtributos_EventosDeLosDispositivos;



NETWORK
TITLE = ---- ---- Recoger el Atributo de los Dispositivos - HORQ
/////////////////////////////////////////////////////////////////////////
/////////////////////////////////////////////////////////////////////////
/////////////////////////////////////////////////////////////////////////
AtributoDeDispositivos_HORQ:NOP   0;
      +AR2  P#5.0;
      TAR2;
      T     #P_Eventos;
      SRD   3;
      T     #OffsetInicial;

// Obtener el Valor del Numero del Dispositivo
      CALL  "FC892_Obtener_ValorDelAtributo"
      ( DB_String := #DBEventosRec,
        OffsetIni := #OffsetInicial,
        Valor     := #ValorDeAtributo
      );
      L     #ValorDeAtributo;  // Lo guardo
      T     #AtributosDeDispositivos.MesaHorquilla;

// Continuo con el Evento
      L     #P_Eventos;
      LAR2;
      JU    InicioBucleAtributos_EventosDeLosDispositivos;



NETWORK
TITLE = ---- ---- Recoger el Atributo de los Dispositivos - POSI
/////////////////////////////////////////////////////////////////////////
/////////////////////////////////////////////////////////////////////////
/////////////////////////////////////////////////////////////////////////
AtributoDeDispositivos_POSI:NOP   0;
      +AR2  P#5.0;
      TAR2;
      T     #P_Eventos;
      SRD   3;
      T     #OffsetInicial;

// Obtener el Valor del Numero del Dispositivo
      CALL  "FC892_Obtener_ValorDelAtributo"
      ( DB_String := #DBEventosRec,
        OffsetIni := #OffsetInicial,
        Valor     := #ValorDeAtributo
      );
      L     #ValorDeAtributo;  // Lo guardo
      T     #AtributosDeDispositivos.MesaCargaDesCarga;

// Continuo con el Evento
      L     #P_Eventos;
      LAR2;
      JU    InicioBucleAtributos_EventosDeLosDispositivos;



NETWORK
TITLE = Distribucion para Guardar Datos del Evento Recibido (LIsta del DB de Conversion) ///////
/////////////////////////////////////////////////////////////////////////
/////////////////////////////////////////////////////////////////////////
/////////////////////////////////////////////////////////////////////////
GuardarDatos_EventosRecibidos:NOP   0;
      TAR2;
      T     #P_Eventos;  // Guardo Por donde voy en la lista de eventos

      L     #NumeroEvento;
      JL    NoExiste_GuardarDatos_Eventos;

      JU    NoExiste_GuardarDatos_Eventos;
      JU    GuardarDatos_EventoRecibido_CREA;  // Evento (01) - CREA
      JU    GuardarDatos_EventoRecibido_RUTA;  // Evento (02) - RUTA
      JU    GuardarDatos_EventoRecibido_DRUT;  // Evento (03) - DRUT
      JU    GuardarDatos_EventoRecibido_RETI;  // Evento (04) - RETI
      JU    GuardarDatos_EventoRecibido_BORR;  // Evento (05) - BORR
      JU    GuardarDatos_EventoRecibido_DATA;  // Evento (06) - DATA
      JU    GuardarDatos_EventoRecibido_Refresco_UT;  // Evento (07) - ?UT?
      JU    GuardarDatos_EventoRecibido_MOVE;  // Evento (08) - MOVE
      JU    GuardarDatos_EventoRecibido_DEMB;  // Evento (09) - DEMB

      JU    GuardarDatos_EventoRecibido_CSTA;  // Evento (10) - CSTA
      JU    GuardarDatos_EventoRecibido_DIDO;  // Evento (11) - DIDO

      JU    NoExiste_GuardarDatos_Eventos;  // Evento (12) - ORDE
      JU    NoExiste_GuardarDatos_Eventos;  // Evento (13) - BOET
      JU    NoExiste_GuardarDatos_Eventos;  // Evento (14) - BOBD
      JU    NoExiste_GuardarDatos_Eventos;  // Evento (15) - RUET
      JU    NoExiste_GuardarDatos_Eventos;  // Evento (16) - RUES
      JU    NoExiste_GuardarDatos_Eventos;  // Evento (17) - INIR

      JU    GuardarDatos_EventoRecibido_Refresco_ST;  // Evento (18) - ?ST?

      JU    NoExiste_GuardarDatos_Eventos;  // Evento (19) - QCRE
      JU    NoExiste_GuardarDatos_Eventos;  // Evento (20) - QPR?

      JU    NoExiste_GuardarDatos_Eventos;  // Evento (21) - CHEQ

/////////////////////////////////////////////////////////////////////////
NoExiste_GuardarDatos_Eventos:NOP   0;
      L     #P_Eventos;  // Recupero por donde voy en la lista de eventos
      LAR2;  // Regreso a buscar el siguiente evento
      JU    FinBucle_EventosRecibidos;



NETWORK
TITLE = ////////////////////////////////////////////////////////////////////////////////////////////////////////////

NETWORK
TITLE = Guardar Datos - Evento CREA - Crear una Nueva UT
// Analisis del evento
//   - Inicializa variables de los atributos del Evento
//   - Buscar Atributos o Final del Evento
//   - Guardar datos del Evento
// Analisis de los atributos del Evento
//   - Mirar que atributo del Evento es
//   - Distribuir a recoger los datos del Evento
//   - Recoger el Atributo McKey
//   - Recoger el Atributo MesaActual
//   - Recoger el Atributo Tipo
//   - Recoger el Atributo Codigo de Barras
//   - Recoger el Atributo Grupo de UT
//   - Recoger el Atributo Cantidad de UT en el Grupo
//   - Recoger el Atributo Orden dentro del grupo
//   - Recoger el Atributo Altura
GuardarDatos_EventoRecibido_CREA:NOP   0;

/////////////////////////////////////////////////////////////////////////
/////////////////////////////////////////////////////////////////////////
/////////////////////////////////////////////////////////////////////////
// --- Guardar Datos del Evento Recibido


/////////////////////////////////////////////////////////////////////////
/////////////////////////////////////////////////////////////////////////
/////////////////////////////////////////////////////////////////////////
// --- Control de la Mesa Actual es correcta
      L     #AtributosDeUTs.MesaActual;  // Ver que mesa es
      L     "CTE_OffsetMesa";
      -I;
      T     #VarTempUTs.MesaActual;

      L     #VarTempUTs.MesaActual;  // Comprobar el numero de mesa
      L     1;  // No menor de 1
      <I;  // No es correcto
      JC    Final_EventoRecibido_CREA;
      L     #VarTempUTs.MesaActual;
      L     "CTE_MaxMesas";  // No mayor que el parametro
      >I;  // No es correcto
      JC    Final_EventoRecibido_CREA;


/////////////////////////////////////////////////////////////////////////
/////////////////////////////////////////////////////////////////////////
/////////////////////////////////////////////////////////////////////////
// --- Control del Mckey es correcto
      L     #AtributosDeUTs.Mckey;  // Se ha recibido Mckey = 0
      L     0;  // No se puede Crear
      ==D;
      JC    Final_EventoRecibido_CREA;


/////////////////////////////////////////////////////////////////////////
/////////////////////////////////////////////////////////////////////////
/////////////////////////////////////////////////////////////////////////
// --- Control del Nuevo Mckey no este en el sistema
// --- Comprobación de DUPLICIDAD
      CALL  "FC720_BuscarUT_EnMesa"
      ( Mckey      := #AtributosDeUTs.Mckey,
        MesaActual := #VarTempUTs.MesaActual,
        NumeroUT   := #VarTempUTs.NumeroUT
      );

      L     #VarTempUTs.NumeroUT;  // Existe UT, Hay DUPLICIDAD de Mckey
      L     0;
      ==I;
      JC    MckeyCorrecto_EventoRecibido_CREA;

// --- Informe de Duplicadad del Mckey
      SET;
      S     "DB812_UTs_Control".UT[#VarTempUTs.NumeroUT].EventosInformarJdT.DuplicidadMckey;

      JU    Final_EventoRecibido_CREA;

MckeyCorrecto_EventoRecibido_CREA:NOP   0;


/////////////////////////////////////////////////////////////////////////
/////////////////////////////////////////////////////////////////////////
/////////////////////////////////////////////////////////////////////////
// --- Control de la Mesa este Definida
      SET;
      AN    "DB850_DefinicionMesas".Mesa[#VarTempUTs.MesaActual].ConfigMesa.MesaPaso;
      AN    "DB850_DefinicionMesas".Mesa[#VarTempUTs.MesaActual].ConfigMesa.MesaCruce;
      AN    "DB850_DefinicionMesas".Mesa[#VarTempUTs.MesaActual].ConfigMesa.MesaMultiplesDestinos;
      JC    Final_EventoRecibido_CREA;


/////////////////////////////////////////////////////////////////////////
/////////////////////////////////////////////////////////////////////////
/////////////////////////////////////////////////////////////////////////
// --- Crear UT en la Mesa Actual
// --- Nota: Rellena ya en UT el Mckey y la Mesa Actual
      CALL  "FC721_CrearUT_EnMesa"
      ( McKey      := #AtributosDeUTs.Mckey,
        MesaActual := #VarTempUTs.MesaActual,
        NumeroUT   := #VarTempUTs.NumeroUT
      );

      L     #VarTempUTs.NumeroUT;
      L     0;  // No se ha podido crear
      ==I;
      JC    Final_EventoRecibido_CREA;



NETWORK
TITLE = ---- Accion del Evento
/////////////////////////////////////////////////////////////////////////
/////////////////////////////////////////////////////////////////////////
/////////////////////////////////////////////////////////////////////////
// --- Guardar datos en la UT, Mckey y Mesa ya estan
      L     202;  // 202 - Recibido Evento de Creada una Nueva UT en la Mesa
      T     "DB812_UTs_Control".UT[#VarTempUTs.NumeroUT].EstadoEventoRecibido;

      L     #AtributosDeUTs.TipoCarga;
      T     "DB812_UTs_Control".UT[#VarTempUTs.NumeroUT].TipoCarga;

      SET;
      A     #AtributosDeUTs.AtributosTipoDeCarga.Pila;
      S     "DB812_UTs_Control".UT[#VarTempUTs.NumeroUT].AtributosDelaCarga.Pila;
      SET;
      A     #AtributosDeUTs.AtributosTipoDeCarga.Remontada;
      S     "DB812_UTs_Control".UT[#VarTempUTs.NumeroUT].AtributosDelaCarga.Remontada;
      SET;
      A     #AtributosDeUTs.AtributosTipoDeCarga.Vacia;
      S     "DB812_UTs_Control".UT[#VarTempUTs.NumeroUT].AtributosDelaCarga.Vacia;


      L     #AtributosDeUTs.GaliboAltura;
      T     "DB815_UTs_Datos".UT[#VarTempUTs.NumeroUT].GaliboAltura;
      L     #AtributosDeUTs.GaliboAnchura;
      T     "DB815_UTs_Datos".UT[#VarTempUTs.NumeroUT].GaliboAnchura;
      L     #AtributosDeUTs.GaliboProfundidad;
      T     "DB815_UTs_Datos".UT[#VarTempUTs.NumeroUT].GaliboProfundidad;

      L     #AtributosDeUTs.GaliboTaco;
      T     "DB815_UTs_Datos".UT[#VarTempUTs.NumeroUT].GaliboTaco;
      L     #AtributosDeUTs.GaliboHueco;
      T     "DB815_UTs_Datos".UT[#VarTempUTs.NumeroUT].GaliboHueco;
      L     #AtributosDeUTs.GaliboHuecoRemontada;
      T     "DB815_UTs_Datos".UT[#VarTempUTs.NumeroUT].GaliboHuecoRemontado;

      L     #AtributosDeUTs.GaliboColor;
      T     "DB815_UTs_Datos".UT[#VarTempUTs.NumeroUT].GaliboColor;
      L     #AtributosDeUTs.GaliboPatin;
      T     "DB815_UTs_Datos".UT[#VarTempUTs.NumeroUT].GaliboPatin;


      L     #AtributosDeUTs.CodigoFlejado;
      T     "DB815_UTs_Datos".UT[#VarTempUTs.NumeroUT].CodigoFlejado;
      L     #AtributosDeUTs.CodigoEnfardado;
      T     "DB815_UTs_Datos".UT[#VarTempUTs.NumeroUT].CodigoEnfardado;
      L     #AtributosDeUTs.CodigoEtiquetado;
      T     "DB815_UTs_Datos".UT[#VarTempUTs.NumeroUT].CodigoEtiquetado;

      L     #AtributosDeUTs.Peso;
      T     "DB815_UTs_Datos".UT[#VarTempUTs.NumeroUT].Peso;

      L     #AtributosDeUTs.CotaAltura;
      T     "DB815_UTs_Datos".UT[#VarTempUTs.NumeroUT].CotaAltura;
      L     #AtributosDeUTs.CotaAnchura;
      T     "DB815_UTs_Datos".UT[#VarTempUTs.NumeroUT].CotaAnchura;
      L     #AtributosDeUTs.CotaProfundidad;
      T     "DB815_UTs_Datos".UT[#VarTempUTs.NumeroUT].CotaProfundidad;

      L     #AtributosDeUTs.CotaAmarre;
      T     "DB815_UTs_Datos".UT[#VarTempUTs.NumeroUT].Amarre;
      L     #AtributosDeUTs.Presion;
      T     "DB815_UTs_Datos".UT[#VarTempUTs.NumeroUT].Presion;

      L     #AtributosDeUTs.Grupo;
      T     "DB812_UTs_Control".UT[#VarTempUTs.NumeroUT].Grupo;
      L     #AtributosDeUTs.CantidadGrupo;
      T     "DB812_UTs_Control".UT[#VarTempUTs.NumeroUT].CantidadGrupo;
      L     #AtributosDeUTs.PosicionGrupo;
      T     "DB812_UTs_Control".UT[#VarTempUTs.NumeroUT].PosicionGrupo;


/////////////////////////////////////////////////////////////////////////
// --- Posicion de la Etiqueta (0) Derecha (1) Izquierdo
      SET;  // Posicion de la Etiqueta
      L     #AtributosDeUTs.PosicionDeLaEtiqueta;
      L     1;  // Lado Derecho = 0
      ==I;
      R     "DB812_UTs_Control".UT[#VarTempUTs.NumeroUT].AtributosDeLaUT.LadoDeLaEtiqueta;

      SET;  // Posicion de la Etiqueta
      L     #AtributosDeUTs.PosicionDeLaEtiqueta;
      L     2;  // Lado Izquierdo = 1
      ==I;
      S     "DB812_UTs_Control".UT[#VarTempUTs.NumeroUT].AtributosDeLaUT.LadoDeLaEtiqueta;


/////////////////////////////////////////////////////////////////////////
// --- Guardar la etiqueta
      CALL  BLKMOV
      ( SRCBLK  := #AtributosDeUTs.Etiqueta,
        RET_VAL := #ReturnValor,
        DSTBLK  := "DB814_UTs_Etiqueta".UT[#VarTempUTs.NumeroUT].Etiqueta
      );

/////////////////////////////////////////////////////////////////////////
// --- Guardar Datos de QUBIQA
      L     #AtributosDeUTs.QUBIQA_NumeroBulto;  // Numero de Bulto
      T     "DB820_UTs_DatosQUBIQA".UT[#VarTempUTs.NumeroUT].NumeroDeBulto;
      L     #AtributosDeUTs.QUBIQA_TotalBultos;  // Numero de Bultos
      T     "DB820_UTs_DatosQUBIQA".UT[#VarTempUTs.NumeroUT].TotalBultos;

      CALL  BLKMOV
      ( SRCBLK  := #AtributosDeUTs.QUBIQA_PID,
        RET_VAL := #ReturnValor,
        DSTBLK  := "DB820_UTs_DatosQUBIQA".UT[#VarTempUTs.NumeroUT].PID
      );  // Guardar el PID


/////////////////////////////////////////////////////////////////////////
// Guardar Ruta si es necesario
// Si hay ruta Nueva - Guardar MesaDestino, Mesa Intermedia y la nueva ruta
      L     0;  // Si existe Nueva Ruta - MesaDestino <> 0
      L     #AtributosDeUTs.MesaDestino;
      ==I;
      JC    FinalGuardarRuta_EventoRecibido_CREA;


/////////////////////////////////////////////////////////////////////////
// Puntero a la UT, Marcar si es necesario -->
//           Actual = Destino = InterMedia --> Marcar la UT
// MODIFICACION --> 06/05/2013 (Alonso)

      SET;  // Reset - Recircular la Carga - Memoria del Retirar
      R     "DB812_UTs_Control".UT[#VarTempUTs.NumeroUT].AtributosDeLaUT.RecircularCarga;
      R     "DB812_UTs_Control".UT[#VarTempUTs.NumeroUT].AtributosDeLaUT.MemorizarRETI;

      L     "DB812_UTs_Control".UT[#VarTempUTs.NumeroUT].MesaActual;
      L     #AtributosDeUTs.MesaDestino;
      <>I;  // MesaActual <> MesaDestino ?
      JC    NoRecirculaLaCarga_EventoRecibido_CREA;

      L     #AtributosDeUTs.MesaDestino;
      L     #AtributosDeUTs.Ruta[0];
      ==I;
      JC    NoRecirculaLaCarga_EventoRecibido_CREA;

      SET;  // Set - Recircular la Carga
      S     "DB812_UTs_Control".UT[#VarTempUTs.NumeroUT].AtributosDeLaUT.RecircularCarga;

NoRecirculaLaCarga_EventoRecibido_CREA:NOP   0;

      L     #AtributosDeUTs.MesaDestino;
      T     "DB812_UTs_Control".UT[#VarTempUTs.NumeroUT].MesaDestino;
      L     #AtributosDeUTs.MesaIntermedia;
      T     "DB812_UTs_Control".UT[#VarTempUTs.NumeroUT].MesaIntermedia;

      CALL  BLKMOV
      ( SRCBLK  := #AtributosDeUTs.Ruta,
        RET_VAL := #ReturnValor,
        DSTBLK  := "DB813_UTs_Ruta".UT[#VarTempUTs.NumeroUT].Ruta
      );

      L     201;  // 201 - Recibido Evento de nueva ruta para la UT
      T     "DB812_UTs_Control".UT[#VarTempUTs.NumeroUT].EstadoEventoRecibido;

//////////////////////////////////////////////////////////////////////
/// Inicio - Realizado 2017 07 06 // Control para Peticion de Ruta
      L     "DB812_UTs_Control".UT[#VarTempUTs.NumeroUT].MesaActual;
      L     #AtributosDeUTs.MesaDestino;
      <>I;
      JC    FinalGuardarRuta_EventoRecibido_CREA;

// Activar la Peticion de RUTA por llegada a su destino
      L     21;  // 21 - Generar Evento Pedir Ruta
      T     "DB812_UTs_Control".UT[#VarTempUTs.NumeroUT].EstadoGeneralUT;
      L     0;  // 0 - No Vale el Evento Recibido
      T     "DB812_UTs_Control".UT[#VarTempUTs.NumeroUT].EstadoEventoRecibido;

//////////////////////////////////////////////////////////////////////
// Final de Guardar Ruta
FinalGuardarRuta_EventoRecibido_CREA:NOP   0;



NETWORK
TITLE = ---- Final
/////////////////////////////////////////////////////////////////////////
/////////////////////////////////////////////////////////////////////////
/////////////////////////////////////////////////////////////////////////
// Se acabo el evento
Final_EventoRecibido_CREA:NOP   0;
      L     #P_Eventos;  // Recupero por donde voy en la lista de eventos
      LAR2;  // Regreso a buscar el siguiente evento
      JU    FinBucle_EventosRecibidos;



NETWORK
TITLE = Guardar Datos - Evento RUTA - Asignar ruta nueva a la UT
// Analisis del evento
//   - Inicializa variables de los atributos del Evento
//   - Buscar Atributos o Final del Evento
//   - Guardar datos del Evento
// Analisis de los atributos del Evento
//   - Mirar que atributo del Evento es
//   - Distribuir a recoger los datos del Evento
//   - Recoger el Atributo McKey
//   - Recoger el Atributo MesaActual
//   - Recoger el Atributo Nueva Ruta
GuardarDatos_EventoRecibido_RUTA:NOP   0;

/////////////////////////////////////////////////////////////////////////
/////////////////////////////////////////////////////////////////////////
/////////////////////////////////////////////////////////////////////////
// --- Guardar Datos del Evento Recibido


/////////////////////////////////////////////////////////////////////////
/////////////////////////////////////////////////////////////////////////
/////////////////////////////////////////////////////////////////////////
// --- Control de la Mesa Actual es Correcta
      L     #AtributosDeUTs.MesaActual;
      L     0;
      ==I;
      JC    FinControlMesa_EventoRecibido_RUTA;

      L     #AtributosDeUTs.MesaActual;  // Ver que mesa es
      L     "CTE_OffsetMesa";
      -I;
      T     #VarTempUTs.MesaActual;

      L     #VarTempUTs.MesaActual;  // Comprobar el numero de mesa
      L     1;  // No menor de 1
      <I;  // No es correcto
      JC    Final_EventoRecibido_RUTA;
      L     #VarTempUTs.MesaActual;
      L     "CTE_MaxMesas";  // No mayor que el parametro
      >I;  // No es correcto
      JC    Final_EventoRecibido_RUTA;

/////////////////////////////////////////////////////////////////////////
FinControlMesa_EventoRecibido_RUTA:NOP   0;


/////////////////////////////////////////////////////////////////////////
/////////////////////////////////////////////////////////////////////////
/////////////////////////////////////////////////////////////////////////
// --- Buscar UT en la Mesa Actual o por Mckey

      CALL  "FC720_BuscarUT_EnMesa"
      ( Mckey      := #AtributosDeUTs.Mckey,
        MesaActual := #VarTempUTs.MesaActual,
        NumeroUT   := #VarTempUTs.NumeroUT
      );

      L     #VarTempUTs.NumeroUT;
      L     0;
      ==I;  // No existe UT
      JC    Final_EventoRecibido_RUTA;



NETWORK
TITLE = ---- Accion del Evento
/////////////////////////////////////////////////////////////////////////
/////////////////////////////////////////////////////////////////////////
/////////////////////////////////////////////////////////////////////////
// Puntero a la UT, Marcar si es necesario -->
//           Actual = Destino = InterMedia --> Marcar la UT
// MODIFICACION --> 06/05/2013 (Alonso)

      SET;  // Reset - Recircular la Carga - Memoria del Retirar
      R     "DB812_UTs_Control".UT[#VarTempUTs.NumeroUT].AtributosDeLaUT.RecircularCarga;
      R     "DB812_UTs_Control".UT[#VarTempUTs.NumeroUT].AtributosDeLaUT.MemorizarRETI;

      L     "DB812_UTs_Control".UT[#VarTempUTs.NumeroUT].MesaActual;
      L     #AtributosDeUTs.MesaDestino;
      <>I;  // MesaActual <> MesaDestino ?
      JC    GuardarRutaRecibida_EventoRecibido_RUTA;

      L     #AtributosDeUTs.MesaDestino;
      L     #AtributosDeUTs.Ruta[0];
      ==I;
      JC    GuardarRutaRecibida_EventoRecibido_RUTA;

      SET;  // Set - Recircular la Carga
      S     "DB812_UTs_Control".UT[#VarTempUTs.NumeroUT].AtributosDeLaUT.RecircularCarga;


/////////////////////////////////////////////////////////////////////////
/////////////////////////////////////////////////////////////////////////
/////////////////////////////////////////////////////////////////////////
// --- Guardar ruta
GuardarRutaRecibida_EventoRecibido_RUTA:NOP   0;

      L     #AtributosDeUTs.MesaDestino;
      T     "DB812_UTs_Control".UT[#VarTempUTs.NumeroUT].MesaDestino;
      L     #AtributosDeUTs.MesaIntermedia;
      T     "DB812_UTs_Control".UT[#VarTempUTs.NumeroUT].MesaIntermedia;

      CALL  BLKMOV
      ( SRCBLK  := #AtributosDeUTs.Ruta,
        RET_VAL := #ReturnValor,
        DSTBLK  := "DB813_UTs_Ruta".UT[#VarTempUTs.NumeroUT].Ruta
      );

      L     201;  // 201 - Recibido Evento de Nueva Ruta para la UT
      T     "DB812_UTs_Control".UT[#VarTempUTs.NumeroUT].EstadoEventoRecibido;


/////////////////////////////////////////////////////////////////////////
/////////////////////////////////////////////////////////////////////////
//////////////////////////////////////////////////////////////////////
/// Inicio - Realizado 2017 07 06 // Control para Peticion de Ruta
      L     "DB812_UTs_Control".UT[#VarTempUTs.NumeroUT].MesaActual;
      L     #AtributosDeUTs.MesaDestino;
      <>I;
      JC    NoPedirRuta_EventoRecibido_RUTA;

      SET;  // Recircular la Carga ?
      A     "DB812_UTs_Control".UT[#VarTempUTs.NumeroUT].AtributosDeLaUT.RecircularCarga;
      JC    NoPedirRuta_EventoRecibido_RUTA;

// Activar la Peticion de RUTA por llegada a su destino
      L     21;  // 21 - Generar Evento Pedir Ruta
      T     "DB812_UTs_Control".UT[#VarTempUTs.NumeroUT].EstadoGeneralUT;
      L     0;  // 0 - No Vale el Evento Recibido
      T     "DB812_UTs_Control".UT[#VarTempUTs.NumeroUT].EstadoEventoRecibido;

//////////////////////////////////////////////////////////////////////
NoPedirRuta_EventoRecibido_RUTA:NOP   0;



NETWORK
TITLE = ---- Final
//////////////////////////////////////////////////////////////////////
//////////////////////////////////////////////////////////////////////
//////////////////////////////////////////////////////////////////////
// --- Se acabo el evento
Final_EventoRecibido_RUTA:NOP   0;
      L     #P_Eventos;  // Recupero por donde voy en la lista de eventos
      LAR2;  // Regreso a buscar el siguiente evento
      JU    FinBucle_EventosRecibidos;



NETWORK
TITLE = Guardar Datos - Evento DRUT - Asignar ruta nueva a la UT (Dinamica)
// Analisis del evento
//   - Inicializa variables de los atributos del Evento
//   - Buscar Atributos o Final del Evento
//   - Guardar datos del Evento
// Analisis de los atributos del Evento
//   - Mirar que atributo del Evento es
//   - Distribuir a recoger los datos del Evento
//   - Recoger el Atributo McKey
//   - Recoger el Atributo MesaActual
//   - Recoger el Atributo Nueva Ruta
GuardarDatos_EventoRecibido_DRUT:NOP   0;

/////////////////////////////////////////////////////////////////////////
/////////////////////////////////////////////////////////////////////////
/////////////////////////////////////////////////////////////////////////
// --- Guardar Datos del Evento Recibido


/////////////////////////////////////////////////////////////////////////
/////////////////////////////////////////////////////////////////////////
/////////////////////////////////////////////////////////////////////////
// --- Control de la Mesa Actual Recibida
      L     #AtributosDeUTs.MesaActual;
      L     0;
      ==I;
      JC    FinControlMesa_EventoRecibido_DRUT;

      L     #AtributosDeUTs.MesaActual;  // Ver que mesa es
      L     "CTE_OffsetMesa";
      -I;
      T     #VarTempUTs.MesaActual;

      L     #VarTempUTs.MesaActual;  // Comprobar el numero de mesa
      L     1;  // No menor de 1
      <I;  // No es correcto
      JC    Final_EventoRecibido_DRUT;
      L     #VarTempUTs.MesaActual;
      L     "CTE_MaxMesas";  // No mayor que el parametro
      >I;  // No es correcto
      JC    Final_EventoRecibido_DRUT;

/////////////////////////////////////////////////////////////////////////
FinControlMesa_EventoRecibido_DRUT:NOP   0;


/////////////////////////////////////////////////////////////////////////
/////////////////////////////////////////////////////////////////////////
/////////////////////////////////////////////////////////////////////////
// --- Buscar UT en la Mesa Actual o por Mckey

      CALL  "FC720_BuscarUT_EnMesa"
      ( Mckey      := #AtributosDeUTs.Mckey,
        MesaActual := #VarTempUTs.MesaActual,
        NumeroUT   := #VarTempUTs.NumeroUT
      );

      L     #VarTempUTs.NumeroUT;
      L     0;  // No existe UT
      ==I;
      JC    Final_EventoRecibido_DRUT;



NETWORK
TITLE = ---- Accion del Evento
/////////////////////////////////////////////////////////////////////////
/////////////////////////////////////////////////////////////////////////
/////////////////////////////////////////////////////////////////////////
// --- Guardar ruta

      L     #AtributosDeUTs.MesaDestino;
      T     "DB812_UTs_Control".UT[#VarTempUTs.NumeroUT].MesaDestino;
      L     #AtributosDeUTs.MesaIntermedia;
      T     "DB812_UTs_Control".UT[#VarTempUTs.NumeroUT].MesaIntermedia;

      CALL  BLKMOV
      ( SRCBLK  := #AtributosDeUTs.Ruta,
        RET_VAL := #ReturnValor,
        DSTBLK  := "DB813_UTs_Ruta".UT[#VarTempUTs.NumeroUT].Ruta
      );



NETWORK
TITLE = ---- Final
//////////////////////////////////////////////////////////////////////
//////////////////////////////////////////////////////////////////////
//////////////////////////////////////////////////////////////////////
// --- Se acabo el evento
Final_EventoRecibido_DRUT:NOP   0;
      L     #P_Eventos;  // Recupero por donde voy en la lista de eventos
      LAR2;  // Regreso a buscar el siguiente evento
      JU    FinBucle_EventosRecibidos;



NETWORK
TITLE = Guardar Datos - Evento RETI - Retirar la UT
// Analisis del evento
//   - Inicializa variables de los atributos del Evento
//   - Buscar Atributos o Final del Evento
//   - Guardar datos del Evento
// Analisis de los atributos del Evento
//   - Mirar que atributo del Evento es
//   - Distribuir a recoger los datos del Evento
//   - Recoger el Atributo McKey
//   - Recoger el Atributo MesaActual
GuardarDatos_EventoRecibido_RETI:NOP   0;

/////////////////////////////////////////////////////////////////////////
/////////////////////////////////////////////////////////////////////////
/////////////////////////////////////////////////////////////////////////
// --- Guardar Datos del Evento Recibido


/////////////////////////////////////////////////////////////////////////
/////////////////////////////////////////////////////////////////////////
/////////////////////////////////////////////////////////////////////////
// --- Control de Mesa Recibida
      L     #AtributosDeUTs.MesaActual;
      L     0;
      ==I;
      JC    FinControlMesa_EventoRecibido_RETI;

      L     #AtributosDeUTs.MesaActual;  // Ver que mesa es
      L     "CTE_OffsetMesa";
      -I;
      T     #VarTempUTs.MesaActual;

      L     #VarTempUTs.MesaActual;  // Comprobar el numero de mesa
      L     1;  // No menor de 1
      <I;  // No es correcto
      JC    Final_EventoRecibido_RETI;
      L     #VarTempUTs.MesaActual;
      L     "CTE_MaxMesas";  // No mayor que el parametro
      >I;  // No es correcto
      JC    Final_EventoRecibido_RETI;

/////////////////////////////////////////////////////////////////////////
FinControlMesa_EventoRecibido_RETI:NOP   0;


/////////////////////////////////////////////////////////////////////////
/////////////////////////////////////////////////////////////////////////
/////////////////////////////////////////////////////////////////////////
// --- Buscar UT en la Mesa Actual o Mckey
      CALL  "FC720_BuscarUT_EnMesa"
      ( Mckey      := #AtributosDeUTs.Mckey,
        MesaActual := #VarTempUTs.MesaActual,
        NumeroUT   := #VarTempUTs.NumeroUT
      );

      L     #VarTempUTs.NumeroUT;
      L     0;  // No existe UT
      ==I;
      JC    Final_EventoRecibido_RETI;



NETWORK
TITLE = ---- Accion del Evento
/////////////////////////////////////////////////////////////////////////
/////////////////////////////////////////////////////////////////////////
/////////////////////////////////////////////////////////////////////////
// --- Guardar datos
      L     #AtributosDeUTs.OrdenSalida;  // Sumar el numero de salida del Atributo
      L     210;  // 210 - Evento de Retirar la UT por S0
      +I;
      T     #VarTempUTs.SalidaEventoRETI;

      SET;  // Memorizar RETI - Ya memorizado
      A     "DB812_UTs_Control".UT[#VarTempUTs.NumeroUT].AtributosDeLaUT.MemorizarRETI;
      JC    ActivadaMemoria_EventoRecibido_RETI;

      L     #VarTempUTs.SalidaEventoRETI;  // EstadoEventoRecibido
      T     "DB812_UTs_Control".UT[#VarTempUTs.NumeroUT].EstadoEventoRecibido;

/////////////////////////////////////////////////////////////////////////
ActivadaMemoria_EventoRecibido_RETI:NOP   0;

      L     #VarTempUTs.SalidaEventoRETI;  // Mesa Intermeria --> Salida RETI
      T     "DB812_UTs_Control".UT[#VarTempUTs.NumeroUT].MesaIntermedia;

      SET;  // Set - Memorizar RETI
      S     "DB812_UTs_Control".UT[#VarTempUTs.NumeroUT].AtributosDeLaUT.MemorizarRETI;



NETWORK
TITLE = ---- Final
/////////////////////////////////////////////////////////////////////////
/////////////////////////////////////////////////////////////////////////
/////////////////////////////////////////////////////////////////////////
// Se acabo el evento
Final_EventoRecibido_RETI:NOP   0;
      L     #P_Eventos;  // Recupero por donde voy en la lista de eventos
      LAR2;  // Regreso a buscar el siguiente evento
      JU    FinBucle_EventosRecibidos;



NETWORK
TITLE = Guardar Datos - Evento BORR - Borrar la UT
// Analisis del evento
//   - Inicializa variables de los atributos del Evento
//   - Buscar Atributos o Final del Evento
//   - Guardar datos del Evento
// Analisis de los atributos del Evento
//   - Mirar que atributo del Evento es
//   - Distribuir a recoger los datos del Evento
//   - Recoger el Atributo McKey
//   - Recoger el Atributo MesaActual
GuardarDatos_EventoRecibido_BORR:NOP   0;

/////////////////////////////////////////////////////////////////////////
/////////////////////////////////////////////////////////////////////////
/////////////////////////////////////////////////////////////////////////
// --- Guardar Datos del Evento Recibido


/////////////////////////////////////////////////////////////////////////
/////////////////////////////////////////////////////////////////////////
/////////////////////////////////////////////////////////////////////////
// --- Control de Mesa Recibida
      L     #AtributosDeUTs.MesaActual;
      L     0;
      ==I;
      JC    FinControlMesa_EventoRecibido_BORR;

      L     #AtributosDeUTs.MesaActual;  // Ver que mesa es
      L     "CTE_OffsetMesa";
      -I;
      T     #VarTempUTs.MesaActual;

      L     #VarTempUTs.MesaActual;  // Comprobar el numero de mesa
      L     1;  // No menor de 1
      <I;  // No es correcto
      JC    Final_EventoRecibido_BORR;
      L     #VarTempUTs.MesaActual;
      L     "CTE_MaxMesas";  // No mayor que el parametro
      >I;  // No es correcto
      JC    Final_EventoRecibido_BORR;

/////////////////////////////////////////////////////////////////////////
FinControlMesa_EventoRecibido_BORR:NOP   0;



NETWORK
TITLE = ---- Accion del Evento --> Distribucion
/////////////////////////////////////////////////////////////////////////
/////////////////////////////////////////////////////////////////////////
/////////////////////////////////////////////////////////////////////////
// --- Distribucion

      L     0;  // Borrar UT en Particular
      L     #AtributosDeUTs.Mckey;
      <>D;
      JC    BorrarUT_EventoRecibido_BORR;

      L     0;  // Borrar UTs de la Mesa
      L     #AtributosDeUTs.MesaActual;
      <>I;
      JC    BorrarUTsDeMesa_EventoRecibido_BORR;

/////////////////////////////////////////////////////////////////////////
// --- Defecto --> Borrar todas las UTs
      JU    BorrarTodasLasUTs_EventoRecibido_BORR;



NETWORK
TITLE = ---- Accion del Evento --> Borrar UT
/////////////////////////////////////////////////////////////////////////
/////////////////////////////////////////////////////////////////////////
/////////////////////////////////////////////////////////////////////////
// --- Borrar una UT en particular
BorrarUT_EventoRecibido_BORR:NOP   0;
      L     #AtributosDeUTs.MesaActual;
      T     #VarTempUTs.MesaActual;
      L     0;  // Comprobar si hay mesa
      ==I;
      JC    BuscarUT_BorrarUT_EventoRecibido_BORR;

      L     #AtributosDeUTs.MesaActual;  // Ver que mesa es
      L     "CTE_OffsetMesa";
      -I;
      T     #VarTempUTs.MesaActual;

      L     #VarTempUTs.MesaActual;  // Comprobar el numero de mesa
      L     1;  // No menor de 1
      <I;  // No es correcto
      JC    Final_EventoRecibido_BORR;
      L     #VarTempUTs.MesaActual;
      L     "CTE_MaxMesas";  // No mayor que el parametro
      >I;  // No es correcto
      JC    Final_EventoRecibido_BORR;

BuscarUT_BorrarUT_EventoRecibido_BORR:NOP   0;

/////////////////////////////////////////////////////////////////////////
// --- Buscar UT en la Mesa Actual o por Mckey

      CALL  "FC720_BuscarUT_EnMesa"
      ( Mckey      := #AtributosDeUTs.Mckey,
        MesaActual := #VarTempUTs.MesaActual,
        NumeroUT   := #VarTempUTs.NumeroUT
      );

      L     #VarTempUTs.NumeroUT;
      L     0;  // No existe UT
      ==I;
      JC    Final_EventoRecibido_BORR;

/////////////////////////////////////////////////////////////////////////
// --- Modificar datos
      L     131;  // 131 - Generar Evento de Borrar UT --> ALONSO(20160525)
      T     "DB812_UTs_Control".UT[#VarTempUTs.NumeroUT].EstadoEventoAGenerar;

      JU    Final_EventoRecibido_BORR;



NETWORK
TITLE = ---- Accion del Evento --> Borrar UTs de la Mesa
/////////////////////////////////////////////////////////////////////////
/////////////////////////////////////////////////////////////////////////
/////////////////////////////////////////////////////////////////////////
// ---- Borrar todas las UT's de la Mesa
BorrarUTsDeMesa_EventoRecibido_BORR:NOP   0;
      L     #AtributosDeUTs.MesaActual;  // Ver que mesa es
      L     "CTE_OffsetMesa";
      -I;
      T     #VarTempUTs.MesaActual;

      L     #VarTempUTs.MesaActual;  // Comprobar el numero de mesa
      L     1;  // No menor de 1
      <I;  // No es correcto
      JC    Final_EventoRecibido_BORR;
      L     #VarTempUTs.MesaActual;
      L     "CTE_MaxMesas";  // No mayor que el parametro
      >I;  // No es correcto
      JC    Final_EventoRecibido_BORR;

      L     "DB810_ColasMesas".Colas[#VarTempUTs.MesaActual].UT_PrimeraMesa;
      T     #VarTempUTs.NumeroUT;


/////////////////////////////////////////////////////////////////////////
/////////////////////////////////////////////////////////////////////////
/////////////////////////////////////////////////////////////////////////
// --- Recorrido de todas la UT de la Mesa
BucleBorrarUTsDeMesa_EventoRecibido_BORR:NOP   0;
      L     #VarTempUTs.NumeroUT;
      L     0;  // No hay mas UT en la Mesa
      ==I;
      JC    Final_EventoRecibido_BORR;

      L     131;  // 131 - Generar Evento de Borrar UT --> ALONSO(20160525)
      T     "DB812_UTs_Control".UT[#VarTempUTs.NumeroUT].EstadoEventoAGenerar;

      L     "DB812_UTs_Control".UT[#VarTempUTs.NumeroUT].UT_SiguienteMesa;
      T     #VarTempUTs.NumeroUT;

/////////////////////////////////////////////////////////////////////////
// Continuo recorriendo todas las UTs de la Mesa
      JU    BucleBorrarUTsDeMesa_EventoRecibido_BORR;



NETWORK
TITLE = ---- Accion del Evento --> Borrar UTs de Todas las Mesas
/////////////////////////////////////////////////////////////////////////
/////////////////////////////////////////////////////////////////////////
/////////////////////////////////////////////////////////////////////////
// Borrar todas las UT's de la Instalacion
BorrarTodasLasUTs_EventoRecibido_BORR:NOP   0;
      L     0;
      T     #IndiceMesa;


/////////////////////////////////////////////////////////////////////////
/////////////////////////////////////////////////////////////////////////
/////////////////////////////////////////////////////////////////////////
// --- Recorrido de todas las Mesas
BucleMesasBorrarTodasLasUTs_EventoRecibido_BORR:NOP   0;
      L     #IndiceMesa;
      L     1;
      +I;
      T     #IndiceMesa;

      L     #IndiceMesa;
      L     "CTE_MaxMesas";
      >I;  // No hay mas mesas en la Instalacion
      JC    Final_EventoRecibido_BORR;


/////////////////////////////////////////////////////////////////////////
// Primera UT de la Mesa

      L     "DB810_ColasMesas".Colas[#IndiceMesa].UT_PrimeraMesa;
      T     #VarTempUTs.NumeroUT;


/////////////////////////////////////////////////////////////////////////
/////////////////////////////////////////////////////////////////////////
/////////////////////////////////////////////////////////////////////////
// --- Recorrido de todas la UT de la Mesa
BucleUTsDeMesaBorrarTodasLasUTs_EventoRecibido_BORR:NOP   0;
      L     #VarTempUTs.NumeroUT;
      L     0;
      ==I;  // No hay mas UT en la Mesa
      JC    BucleMesasBorrarTodasLasUTs_EventoRecibido_BORR;

      L     131;  // 131 - Generar Evento de Borrar UT --> ALONSO(20160525)
      T     "DB812_UTs_Control".UT[#VarTempUTs.NumeroUT].EstadoEventoAGenerar;

      L     "DB812_UTs_Control".UT[#VarTempUTs.NumeroUT].UT_SiguienteMesa;
      T     #VarTempUTs.NumeroUT;

// Continuo recorriendo de las UTs de la Mesa
      JU    BucleUTsDeMesaBorrarTodasLasUTs_EventoRecibido_BORR;



NETWORK
TITLE = ---- Final
/////////////////////////////////////////////////////////////////////////
/////////////////////////////////////////////////////////////////////////
/////////////////////////////////////////////////////////////////////////
// Se acabo el evento
Final_EventoRecibido_BORR:NOP   0;
      L     #P_Eventos;  // Recupero por donde voy en la lista de eventos
      LAR2;  // Regreso a buscar el siguiente evento
      JU    FinBucle_EventosRecibidos;



NETWORK
TITLE = Guardar Datos - Evento DATA - Notificacion de Datos de la UT
// Analizar el evento
// - Inicializa variables de los atributos del Evento
// - Buscar Atributos o Final del Evento
// - Guardar datos del Evento
// Analizar atributos del Evento
// - Distribuir a recoger los datos del Evento
// - Recoger el Atributo McKey
// - Recoger el Atributo MesaActual
// - Recoger el Atributo Tipo
// - Recoger el Atributo Codigo de Barras
// - Recoger el Atributo Grupo de UT
// - Recoger el Atributo Cantidad de UT en el Grupo
// - Recoger el Atributo Orden dentro del grupo
// - Recoger el Atributo Altura
GuardarDatos_EventoRecibido_DATA:NOP   0;

/////////////////////////////////////////////////////////////////////////
/////////////////////////////////////////////////////////////////////////
/////////////////////////////////////////////////////////////////////////
// --- Guardar Datos del Evento Recibido


/////////////////////////////////////////////////////////////////////////
/////////////////////////////////////////////////////////////////////////
/////////////////////////////////////////////////////////////////////////
// --- Control de Mesa Recibida
      L     #AtributosDeUTs.MesaActual;
      L     0;
      ==I;
      JC    FinControlMesa_DATA_EventosRecibidos;

      L     #AtributosDeUTs.MesaActual;  // Ver que mesa es
      L     "CTE_OffsetMesa";
      -I;
      T     #VarTempUTs.MesaActual;

      L     #VarTempUTs.MesaActual;  // Comprobar el numero de mesa
      L     1;  // No menor de 1
      <I;  // No es correcto
      JC    Final_EventoRecibido_DATA;  // No es correcto
      L     #VarTempUTs.MesaActual;
      L     "CTE_MaxMesas";  // No meyor que el parametro
      >I;  // No es correcto
      JC    Final_EventoRecibido_DATA;

/////////////////////////////////////////////////////////////////////////
FinControlMesa_DATA_EventosRecibidos:NOP   0;


/////////////////////////////////////////////////////////////////////////
/////////////////////////////////////////////////////////////////////////
/////////////////////////////////////////////////////////////////////////
// ---  Buscar UT, para guardar datos
      CALL  "FC720_BuscarUT_EnMesa"
      ( Mckey      := #AtributosDeUTs.Mckey,
        MesaActual := #VarTempUTs.MesaActual,
        NumeroUT   := #VarTempUTs.NumeroUT
      );

      L     #VarTempUTs.NumeroUT;
      L     0;
      ==I;  // No existe UT, no se hace por ahora
      JC    Final_EventoRecibido_DATA;



NETWORK
TITLE = ----
/////////////////////////////////////////////////////////////////////////
/////////////////////////////////////////////////////////////////////////
/////////////////////////////////////////////////////////////////////////
// --- Avisar de Evento Recibido

      L     204;  // 204 - Recibido Evento de Datos Nuevos de la UT
      T     "DB812_UTs_Control".UT[#VarTempUTs.NumeroUT].EstadoEventoRecibido;


/////////////////////////////////////////////////////////////////////////
/////////////////////////////////////////////////////////////////////////
/////////////////////////////////////////////////////////////////////////
// --- Guardar los datos de TipoCarga
      L     #AtributosDeUTs.TipoCarga;
      L     0;
      ==I;  // No hay que Cambiar el Tipo de Paleta ?
      JC    SinDatosTipoCarga_EventoRecibido_DATA;

      L     #AtributosDeUTs.TipoCarga;
      T     "DB812_UTs_Control".UT[#VarTempUTs.NumeroUT].TipoCarga;

      SET;
      R     "DB812_UTs_Control".UT[#VarTempUTs.NumeroUT].AtributosDelaCarga.Pila;
      R     "DB812_UTs_Control".UT[#VarTempUTs.NumeroUT].AtributosDelaCarga.Remontada;
      R     "DB812_UTs_Control".UT[#VarTempUTs.NumeroUT].AtributosDelaCarga.Vacia;

      SET;
      A     #AtributosDeUTs.AtributosTipoDeCarga.Pila;
      S     "DB812_UTs_Control".UT[#VarTempUTs.NumeroUT].AtributosDelaCarga.Pila;
      SET;
      A     #AtributosDeUTs.AtributosTipoDeCarga.Remontada;
      S     "DB812_UTs_Control".UT[#VarTempUTs.NumeroUT].AtributosDelaCarga.Remontada;
      SET;
      A     #AtributosDeUTs.AtributosTipoDeCarga.Vacia;
      S     "DB812_UTs_Control".UT[#VarTempUTs.NumeroUT].AtributosDelaCarga.Vacia;
SinDatosTipoCarga_EventoRecibido_DATA:NOP   0;


//////////////////////////////////////////////////////////////////////
//////////////////////////////////////////////////////////////////////
//////////////////////////////////////////////////////////////////////
// --- Se cambia todo lo relacionado con el gálibo
      L     #AtributosDeUTs.GaliboAltura;
      L     0;
      ==I;  // No hay que Cambiar la Altura ?
      JC    SinDatosGaliboAltura_EventoRecibido_DATA;

      L     #AtributosDeUTs.GaliboAltura;
      T     "DB815_UTs_Datos".UT[#VarTempUTs.NumeroUT].GaliboAltura;
SinDatosGaliboAltura_EventoRecibido_DATA:NOP   0;

//////////////////////////////////////////////////////////////////////
      L     #AtributosDeUTs.GaliboAnchura;
      L     0;
      ==I;  // No hay que Cambiar la Anchura ?
      JC    SinDatosGaliboAnchura_EventoRecibido_DATA;

      L     #AtributosDeUTs.GaliboAnchura;
      T     "DB815_UTs_Datos".UT[#VarTempUTs.NumeroUT].GaliboAnchura;
SinDatosGaliboAnchura_EventoRecibido_DATA:NOP   0;

//////////////////////////////////////////////////////////////////////
      L     #AtributosDeUTs.GaliboProfundidad;
      L     0;
      ==I;  // No hay que Cambiar la Profundidad ?
      JC    SinDatosGaliboProfundidad_EventoRecibido_DATA;

      L     #AtributosDeUTs.GaliboProfundidad;
      T     "DB815_UTs_Datos".UT[#VarTempUTs.NumeroUT].GaliboProfundidad;
SinDatosGaliboProfundidad_EventoRecibido_DATA:NOP   0;

//////////////////////////////////////////////////////////////////////
      L     #AtributosDeUTs.GaliboHueco;
      L     0;
      ==I;  // No hay que Cambiar la Hueco ?
      JC    SinDatosGaliboHueco_EventoRecibido_DATA;

      L     #AtributosDeUTs.GaliboHueco;
      T     "DB815_UTs_Datos".UT[#VarTempUTs.NumeroUT].GaliboHueco;
SinDatosGaliboHueco_EventoRecibido_DATA:NOP   0;

//////////////////////////////////////////////////////////////////////
      L     #AtributosDeUTs.GaliboTaco;
      L     0;
      ==I;  // No hay que Cambiar la Taco ?
      JC    SinDatosGaliboTaco_EventoRecibido_DATA;

      L     #AtributosDeUTs.GaliboTaco;
      T     "DB815_UTs_Datos".UT[#VarTempUTs.NumeroUT].GaliboTaco;
SinDatosGaliboTaco_EventoRecibido_DATA:NOP   0;

//////////////////////////////////////////////////////////////////////
      L     #AtributosDeUTs.GaliboHuecoRemontada;
      L     0;
      ==I;  // No hay que Cambiar la Hueco Remontada ?
      JC    SinDatosGaliboHuecoRemontada_EventoRecibido_DATA;

      L     #AtributosDeUTs.GaliboHuecoRemontada;
      T     "DB815_UTs_Datos".UT[#VarTempUTs.NumeroUT].GaliboHuecoRemontado;
SinDatosGaliboHuecoRemontada_EventoRecibido_DATA:NOP   0;


//////////////////////////////////////////////////////////////////////
      L     #AtributosDeUTs.GaliboColor;
      L     0;
      ==I;  // No hay que Cambiar la Color ?
      JC    SinDatosGaliboColor_EventoRecibido_DATA;

      L     #AtributosDeUTs.GaliboHuecoRemontada;
      T     "DB815_UTs_Datos".UT[#VarTempUTs.NumeroUT].GaliboColor;
SinDatosGaliboColor_EventoRecibido_DATA:NOP   0;

//////////////////////////////////////////////////////////////////////
      L     #AtributosDeUTs.GaliboPatin;
      L     0;
      ==I;  // No hay que Cambiar la Patin ?
      JC    SinDatosGaliboPatin_EventoRecibido_DATA;

      L     #AtributosDeUTs.GaliboPatin;
      T     "DB815_UTs_Datos".UT[#VarTempUTs.NumeroUT].GaliboPatin;
SinDatosGaliboPatin_EventoRecibido_DATA:NOP   0;







//////////////////////////////////////////////////////////////////////
      L     #AtributosDeUTs.CodigoFlejado;
      L     -1;
      ==I;  // No hay que Cambiar el Flejado ?
      JC    SinDatosCodigoFlejado_EventoRecibido_DATA;

      L     #AtributosDeUTs.CodigoFlejado;
      T     "DB815_UTs_Datos".UT[#VarTempUTs.NumeroUT].CodigoFlejado;
SinDatosCodigoFlejado_EventoRecibido_DATA:NOP   0;


//////////////////////////////////////////////////////////////////////
      L     #AtributosDeUTs.CodigoEnfardado;
      L     -1;
      ==I;  // No hay que Cambiar el Enfardado ?
      JC    SinDatosCodigoEnfardado_EventoRecibido_DATA;

      L     #AtributosDeUTs.CodigoEnfardado;
      T     "DB815_UTs_Datos".UT[#VarTempUTs.NumeroUT].CodigoEnfardado;
SinDatosCodigoEnfardado_EventoRecibido_DATA:NOP   0;


//////////////////////////////////////////////////////////////////////
      L     #AtributosDeUTs.CodigoEtiquetado;
      L     -1;
      ==I;  // No hay que Cambiar el Etiquetado ?
      JC    SinDatosCodigoEtiquetado_EventoRecibido_DATA;

      L     #AtributosDeUTs.CodigoEtiquetado;
      T     "DB815_UTs_Datos".UT[#VarTempUTs.NumeroUT].CodigoEtiquetado;
SinDatosCodigoEtiquetado_EventoRecibido_DATA:NOP   0;


//////////////////////////////////////////////////////////////////////
      L     #AtributosDeUTs.Peso;
      L     0;
      ==I;  // No hay que Cambiar el Peso ?
      JC    SinDatosPeso_EventoRecibido_DATA;

      L     #AtributosDeUTs.Peso;
      T     "DB815_UTs_Datos".UT[#VarTempUTs.NumeroUT].Peso;
SinDatosPeso_EventoRecibido_DATA:NOP   0;


//////////////////////////////////////////////////////////////////////
      L     #AtributosDeUTs.CotaAltura;
      L     0;
      ==I;  // No hay que Cambiar el Altura (Cota) ?
      JC    SinDatosCotaAltura_EventoRecibido_DATA;

      L     #AtributosDeUTs.CotaAltura;
      T     "DB815_UTs_Datos".UT[#VarTempUTs.NumeroUT].CotaAltura;
SinDatosCotaAltura_EventoRecibido_DATA:NOP   0;


//////////////////////////////////////////////////////////////////////
      L     #AtributosDeUTs.CotaAnchura;
      L     0;
      ==I;  // No hay que Cambiar el Cota Anchura ?
      JC    SinDatosCotaAnchura_EventoRecibido_DATA;

      L     #AtributosDeUTs.CotaAnchura;
      T     "DB815_UTs_Datos".UT[#VarTempUTs.NumeroUT].CotaAnchura;
SinDatosCotaAnchura_EventoRecibido_DATA:NOP   0;


//////////////////////////////////////////////////////////////////////
      L     #AtributosDeUTs.CotaProfundidad;
      L     0;
      ==I;  // No hay que Cambiar el Cota Largura ?
      JC    SinDatosCotaProfundidad_EventoRecibido_DATA;

      L     #AtributosDeUTs.CotaProfundidad;
      T     "DB815_UTs_Datos".UT[#VarTempUTs.NumeroUT].CotaProfundidad;
SinDatosCotaProfundidad_EventoRecibido_DATA:NOP   0;


//////////////////////////////////////////////////////////////////////
      L     #AtributosDeUTs.CotaAmarre;
      L     0;
      ==I;  // No hay que Cambiar el Amarre ?
      JC    SinDatosCotaAmarre_EventoRecibido_DATA;

      L     #AtributosDeUTs.CotaAmarre;
      T     "DB815_UTs_Datos".UT[#VarTempUTs.NumeroUT].Amarre;
SinDatosCotaAmarre_EventoRecibido_DATA:NOP   0;


//////////////////////////////////////////////////////////////////////
      L     #AtributosDeUTs.Presion;
      L     0;
      ==I;  // No hay que Cambiar el Presion ?
      JC    SinDatosPresion_EventoRecibido_DATA;

      L     #AtributosDeUTs.Presion;
      T     "DB815_UTs_Datos".UT[#VarTempUTs.NumeroUT].Presion;
SinDatosPresion_EventoRecibido_DATA:NOP   0;


//////////////////////////////////////////////////////////////////////
//////////////////////////////////////////////////////////////////////
//////////////////////////////////////////////////////////////////////
// --- Guardar Grupo
      L     #AtributosDeUTs.Grupo;
      L     0;
      ==I;  // No hay que Cambiar el Grupo ?
      JC    SinDatosGrupo_EventoRecibido_DATA;

      L     #AtributosDeUTs.Grupo;
      T     "DB812_UTs_Control".UT[#VarTempUTs.NumeroUT].Grupo;
      L     #AtributosDeUTs.CantidadGrupo;
      T     "DB812_UTs_Control".UT[#VarTempUTs.NumeroUT].CantidadGrupo;
      L     #AtributosDeUTs.PosicionGrupo;
      T     "DB812_UTs_Control".UT[#VarTempUTs.NumeroUT].PosicionGrupo;
SinDatosGrupo_EventoRecibido_DATA:NOP   0;


//////////////////////////////////////////////////////////////////////
//////////////////////////////////////////////////////////////////////
//////////////////////////////////////////////////////////////////////
// --- Guardar Posicion de la etiqueta

      L     #AtributosDeUTs.PosicionDeLaEtiqueta;  // Posicion de la Etiqueta
      L     1;  // Lado Derecho = 1
      ==I;
      R     "DB812_UTs_Control".UT[#VarTempUTs.NumeroUT].AtributosDeLaUT.LadoDeLaEtiqueta;

      L     #AtributosDeUTs.PosicionDeLaEtiqueta;  // Posicion de la Etiqueta
      L     2;  // Lado Izquierdo = 2
      ==I;
      S     "DB812_UTs_Control".UT[#VarTempUTs.NumeroUT].AtributosDeLaUT.LadoDeLaEtiqueta;


//////////////////////////////////////////////////////////////////////
//////////////////////////////////////////////////////////////////////
//////////////////////////////////////////////////////////////////////
// --- Guardar la Etiqueta

      L     0;
      L     #AtributosDeUTs.Etiqueta[0];
      ==I;
      JC    SinDatosEtiqueta_EventoRecibido_DATA;

      CALL  BLKMOV
      ( SRCBLK  := #AtributosDeUTs.Etiqueta,
        RET_VAL := #ReturnValor,
        DSTBLK  := "DB814_UTs_Etiqueta".UT[#VarTempUTs.NumeroUT].Etiqueta
      );
SinDatosEtiqueta_EventoRecibido_DATA:NOP   0;


//////////////////////////////////////////////////////////////////////
//////////////////////////////////////////////////////////////////////
//////////////////////////////////////////////////////////////////////
// --- Guardar Datos de QUBIQA
      L     0;
      L     #AtributosDeUTs.QUBIQA_NumeroBulto;
      ==I;
      JC    SinDatosQUBIQA_EventoRecibido_DATA;

      L     #AtributosDeUTs.QUBIQA_NumeroBulto;  // Numero de Bulto
      T     "DB820_UTs_DatosQUBIQA".UT[#VarTempUTs.NumeroUT].NumeroDeBulto;
      L     #AtributosDeUTs.QUBIQA_TotalBultos;  // Numero de Bultos
      T     "DB820_UTs_DatosQUBIQA".UT[#VarTempUTs.NumeroUT].TotalBultos;

      CALL  BLKMOV
      ( SRCBLK  := #AtributosDeUTs.QUBIQA_PID,
        RET_VAL := #ReturnValor,
        DSTBLK  := "DB820_UTs_DatosQUBIQA".UT[#VarTempUTs.NumeroUT].PID
      );  // Guardar el PID

SinDatosQUBIQA_EventoRecibido_DATA:NOP   0;



NETWORK
TITLE = ---- Final
//////////////////////////////////////////////////////////////////////
//////////////////////////////////////////////////////////////////////
//////////////////////////////////////////////////////////////////////
// Se acabo el evento
Final_EventoRecibido_DATA:NOP   0;
      L     #P_Eventos;  // Recupero por donde voy en la lista de eventos
      LAR2;
      JU    FinBucle_EventosRecibidos;  // Regreso a buscar el siguiente evento



NETWORK
TITLE = Guardar Datos - Evento ?UT? - Peticion de Refresco de datos de las UT's
// Analisis del Evento
// - Inicializa variables de los atributos del Evento
// - Buscar Atributos o Final del Evento
// - Guardar datos del Evento
//   - Si es UT determinada
//   - Si es una mesa determinada
//   - Si son todas
// Analisis de los atributos del Evento
// - Mirar que atributo del Evento es
// - Distribuir a recoger los datos del Evento
// - Recoger el Atributo McKey
// - Recoger el Atributo MesaActual
GuardarDatos_EventoRecibido_Refresco_UT:NOP   0;

/////////////////////////////////////////////////////////////////////////
/////////////////////////////////////////////////////////////////////////
/////////////////////////////////////////////////////////////////////////
// --- Guardar Datos del Evento Recibido


/////////////////////////////////////////////////////////////////////////
/////////////////////////////////////////////////////////////////////////
/////////////////////////////////////////////////////////////////////////
// --- Control de la Mesa Recibida
      L     #AtributosDeUTs.MesaActual;  // Si ha llegado atributo de Mesa
      L     0;  // Antes de comprobar si es el correcto
      ==I;  // No ha llegado
      JC    FinControlMesa_RefrescoUT_EventosRecibidos;

      L     #AtributosDeUTs.MesaActual;  // Ver que mesa es
      L     "CTE_OffsetMesa";
      -I;
      T     #VarTempUTs.MesaActual;

      L     #VarTempUTs.MesaActual;  // Comprobar el numero de mesa
      L     1;  // No menor de 1
      <I;  // No es correcto
      JC    Final_EventoRecibido_RefrescoUT;
      L     #VarTempUTs.MesaActual;
      L     "CTE_MaxMesas";  // No meyor que el parametro
      >I;  // No es correcto
      JC    Final_EventoRecibido_RefrescoUT;

/////////////////////////////////////////////////////////////////////////
FinControlMesa_RefrescoUT_EventosRecibidos:NOP   0;



NETWORK
TITLE = ---- Accion del Evento --> Distribucion
/////////////////////////////////////////////////////////////////////////
/////////////////////////////////////////////////////////////////////////
/////////////////////////////////////////////////////////////////////////
// --- Distribucion para la busqueda

      L     #AtributosDeUTs.Mckey;
      L     0;
      <>I;  // Es una UT Especifica
      JC    RefrescoDeUT_EventoRecibido_RefrescoUT;

      L     #AtributosDeUTs.MesaActual;
      L     0;
      <>I;  // Son todas las UT de una Mesa
      JC    RefrescoDeUTsDeLaMesa_EventoRecibido_RefrescoUT;

/////////////////////////////////////////////////////////////////////////
// --- Son todas las UT -> Por defecto
      JU    RefrescoDeUTsTodasLasMesas_EventoRecibido_RefrescoUT;



NETWORK
TITLE = ---- Accion del Evento --> Peticion de Refesco de una UT especifica
/////////////////////////////////////////////////////////////////////////
/////////////////////////////////////////////////////////////////////////
/////////////////////////////////////////////////////////////////////////
// Es una UT Especifica
RefrescoDeUT_EventoRecibido_RefrescoUT:NOP   0;
      L     #AtributosDeUTs.MesaActual;
      T     #VarTempUTs.MesaActual;
      L     0;  // Comprobar si hay mesa
      ==I;
      JC    BuscarUT_RefrescoDeUT_EventoRecibido_RefrescoUT;

      L     #AtributosDeUTs.MesaActual;  // Ver que mesa es
      L     "CTE_OffsetMesa";
      -I;
      T     #VarTempUTs.MesaActual;

      L     #VarTempUTs.MesaActual;  // Comprobar el numero de mesa
      L     1;  // No menor de 1
      <I;  // No es correcto
      JC    Final_EventoRecibido_RefrescoUT;
      L     #VarTempUTs.MesaActual;
      L     "CTE_MaxMesas";  // No mayor que el parametro
      >I;  // No es correcto
      JC    Final_EventoRecibido_RefrescoUT;

BuscarUT_RefrescoDeUT_EventoRecibido_RefrescoUT:NOP   0;
      CALL  "FC720_BuscarUT_EnMesa"
      ( Mckey      := #AtributosDeUTs.Mckey,
        MesaActual := #VarTempUTs.MesaActual,
        NumeroUT   := #VarTempUTs.NumeroUT  // Donde esta la UT
      );  // Busca por Mesa o por Mckey

      L     #VarTempUTs.NumeroUT;
      L     0;
      ==I;  // No existe UT, no se hace por ahora
      JC    Final_EventoRecibido_RefrescoUT;


/////////////////////////////////////////////////////////////////////////
/// Generar Peticion de Datos de la UT
// 205 - Recibido Evento de Refesco de datos para la UT (Anulado)
// 22  - Estado General UT Peticion de Refresco de datos

// 2023 01 05 - Anulado >>> Cambio de Sistema
//      L     22                   // 22 - Peticion de Refresco de datos
//      T     "DB812_UTs_Control".UT[#VarTempUTs.NumeroUT].EstadoGeneralUT
// 2023 01 05 - Bits para informar >>> Nueco Sistema
      SET;
      =     "DB812_UTs_Control".UT[#VarTempUTs.NumeroUT].EventosInformarJdT.PeticionDeDatos;

      JU    Final_EventoRecibido_RefrescoUT;



NETWORK
TITLE = ---- Accion del Evento --> Peticion de Refesco de las UTs de una Mesa
/////////////////////////////////////////////////////////////////////////
/////////////////////////////////////////////////////////////////////////
/////////////////////////////////////////////////////////////////////////
// --- Son todas las UT de una Mesa
RefrescoDeUTsDeLaMesa_EventoRecibido_RefrescoUT:NOP   0;
      L     #AtributosDeUTs.MesaActual;  // Ver que mesa es
      L     "CTE_OffsetMesa";
      -I;
      T     #VarTempUTs.MesaActual;

      L     #VarTempUTs.MesaActual;  // Comprobar el numero de mesa
      L     1;  // No menor de 1
      <I;  // No es correcto
      JC    Final_EventoRecibido_RefrescoUT;
      L     #VarTempUTs.MesaActual;
      L     "CTE_MaxMesas";  // No mayor que el parametro
      >I;  // No es correcto
      JC    Final_EventoRecibido_RefrescoUT;

/////////////////////////////////////////////////////////////////////////
/// --- Mirar si esta definido como mesa de tracking
      SET;
      AN    "DB850_DefinicionMesas".Mesa[#VarTempUTs.MesaActual].ConfigMesa.MesaPaso;
      AN    "DB850_DefinicionMesas".Mesa[#VarTempUTs.MesaActual].ConfigMesa.MesaCruce;
      AN    "DB850_DefinicionMesas".Mesa[#VarTempUTs.MesaActual].ConfigMesa.MesaMultiplesDestinos;
      JC    Final_EventoRecibido_RefrescoUT;


/////////////////////////////////////////////////////////////////////////
/// --- Mirar Si pertenece al JDT // JDT01 ?
      SET;
      X     "DB850_DefinicionMesas".Mesa[#VarTempUTs.MesaActual].ConfigMesa.MesaDeJDT02;
      XN    #JDT02_Activo;
      =     #MesaDeJDT02;

      SET;
      AN    #MesaDeJDT02;
      JC    Final_EventoRecibido_RefrescoUT;


/////////////////////////////////////////////////////////////////////////
// --- Primera UT de la Mesa
      L     "DB810_ColasMesas".Colas[#VarTempUTs.MesaActual].UT_PrimeraMesa;
      T     #VarTempUTs.NumeroUT;


/////////////////////////////////////////////////////////////////////////
/////////////////////////////////////////////////////////////////////////
/////////////////////////////////////////////////////////////////////////
BucleRefrescoUTsDeMesa_EventoRecibido_RefrescoUT:NOP   0;
      L     #VarTempUTs.NumeroUT;  // Recorrido de todas la UT de la Mesa
      L     0;
      ==I;  // No hay mas UT en la Mesa
      JC    Final_EventoRecibido_RefrescoUT;

/////////////////////////////////////////////////////////////////////////
/// Generar Peticion de Datos de la UT
// 205 - Recibido Evento de Refesco de datos para la UT (Anulado)
// 22  - Estado General UT Peticion de Refresco de datos

// 2023 01 05 - Anulado >>> Cambio de Sistema
//      L     22                   // 22 - Peticion de Refresco de datos
//      T     "DB812_UTs_Control".UT[#VarTempUTs.NumeroUT].EstadoGeneralUT
// 2023 01 05 - Bits para informar >>> Nueco Sistema
      SET;
      =     "DB812_UTs_Control".UT[#VarTempUTs.NumeroUT].EventosInformarJdT.PeticionDeDatos;

/////////////////////////////////////////////////////////////////////////
// --- Continuo recorriendo la Mesa
      L     "DB812_UTs_Control".UT[#VarTempUTs.NumeroUT].UT_SiguienteMesa;
      T     #VarTempUTs.NumeroUT;
      JU    BucleRefrescoUTsDeMesa_EventoRecibido_RefrescoUT;



NETWORK
TITLE = ---- Accion del Evento --> Peticion de Refesco de las UTs de Todas las Mesas
/////////////////////////////////////////////////////////////////////////
/////////////////////////////////////////////////////////////////////////
/////////////////////////////////////////////////////////////////////////
// --- Son todas las UT de la Instalacion
RefrescoDeUTsTodasLasMesas_EventoRecibido_RefrescoUT:NOP   0;

      L     0;
      T     #IndiceMesa;

/////////////////////////////////////////////////////////////////////////
/////////////////////////////////////////////////////////////////////////
/////////////////////////////////////////////////////////////////////////
// --- Recorrido de todas las Mesas
BucleMesaRefrescoUTsDeMesa_EventoRecibido_RefrescoUT:NOP   0;
      L     #IndiceMesa;
      L     1;
      +I;
      T     #IndiceMesa;

      L     #IndiceMesa;
      L     "CTE_MaxMesas";
      >I;  // No hay mas mesas en la Instalacion
      JC    Final_EventoRecibido_RefrescoUT;


/////////////////////////////////////////////////////////////////////////
/// --- Mirar si esta definido como mesa de tracking
      SET;
      AN    "DB850_DefinicionMesas".Mesa[#IndiceMesa].ConfigMesa.MesaPaso;
      AN    "DB850_DefinicionMesas".Mesa[#IndiceMesa].ConfigMesa.MesaCruce;
      AN    "DB850_DefinicionMesas".Mesa[#IndiceMesa].ConfigMesa.MesaMultiplesDestinos;
      JC    BucleMesaRefrescoUTsDeMesa_EventoRecibido_RefrescoUT;


/////////////////////////////////////////////////////////////////////////
/// --- Mirar Si pertenece al JDT
      SET;
      X     "DB850_DefinicionMesas".Mesa[#IndiceMesa].ConfigMesa.MesaDeJDT02;  // JDT01 ?
      XN    #JDT02_Activo;
      =     #MesaDeJDT02;

      SET;
      AN    #MesaDeJDT02;
      JC    BucleMesaRefrescoUTsDeMesa_EventoRecibido_RefrescoUT;


/////////////////////////////////////////////////////////////////////////
/////////////////////////////////////////////////////////////////////////
/////////////////////////////////////////////////////////////////////////
// --- Recorrer la Mesa

      L     "DB810_ColasMesas".Colas[#IndiceMesa].UT_PrimeraMesa;
      T     #VarTempUTs.NumeroUT;

BucleUTsMesaRefrescoUTsDeMesa_EventoRecibido_RefrescoUT:NOP   0;
      L     #VarTempUTs.NumeroUT;  // Recorrido de todas la UT de la Mesa
      L     0;
      ==I;  // No hay mas UT en la Mesa
      JC    BucleMesaRefrescoUTsDeMesa_EventoRecibido_RefrescoUT;

/////////////////////////////////////////////////////////////////////////
/// --- Generar Peticion de Datos de la UT
// 205 - Recibido Evento de Refesco de datos para la UT (Anulado)
// 22  - Estado General UT Peticion de Refresco de datos

// 2023 01 05 - Anulado >>> Cambio de Sistema
//      L     22                   // 22 - Peticion de Refresco de datos
//      T     "DB812_UTs_Control".UT[#VarTempUTs.NumeroUT].EstadoGeneralUT
// 2023 01 05 - Bits para informar >>> Nueco Sistema
      SET;
      =     "DB812_UTs_Control".UT[#VarTempUTs.NumeroUT].EventosInformarJdT.PeticionDeDatos;

/////////////////////////////////////////////////////////////////////////
// --- Continuo recorriendo la Mesa
      L     "DB812_UTs_Control".UT[#VarTempUTs.NumeroUT].UT_SiguienteMesa;
      T     #VarTempUTs.NumeroUT;
      JU    BucleUTsMesaRefrescoUTsDeMesa_EventoRecibido_RefrescoUT;



